KUKA KRL program: MyProgram_039().src

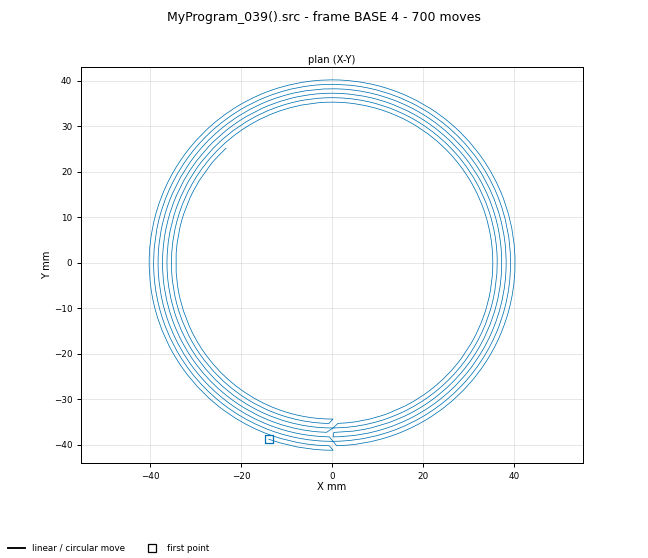
[picture p0: tool path of MyProgram_039().src in frame BASE 4, 700 of 700 moves have a stored position in this frame; points joined in program order, loops and branches not executed]
&ACCESS RVP
&REL 1
&PARAM TEMPLATE = C:\KRC\Roboter\Template\vorgabe
&PARAM EDITMASK = *
DEF MyProgram_039()
; ---- Setting reference (Base) ----
$BASE = BASE_DATA[4]

; --------------------------
; ---- Setting tool (TCP) ----
$TOOL = TOOL_DATA[3]
; --------------------------

$VEL.CP = VEL_APROX_PRINT
Startdeposition()
$VEL.CP = VEL_PRINT
LIN {X -13.9314,Y -38.786,Z 62,A -114.6314,B 24.865,C -2.6814,E1 24.9501,E2 -882.0703} C_DIS
LIN {X -11.5629,Y -39.5572,Z 62,A -111.3021,B 24.8654,C -2.6773,E1 24.959,E2 -885.3951} C_DIS
LIN {X -7.6518,Y -40.4959,Z 62,A -105.6604,B 24.8656,C -2.6755,E1 24.9744,E2 -891.0395} C_DIS
LIN {X -3.6812,Y -41.0476,Z 62,A -101.0464,B 24.867,C -2.6611,E1 24.9871,E2 -895.6225} C_DIS
LIN {X -1.5443,Y -41.1835,Z 62,A -97.4937,B 24.8662,C -2.6695,E1 24.9971,E2 -899.1962} C_DIS
LIN {X 0.2272,Y -41.2107,Z 62,A -96.0828,B 24.8676,C -2.6549,E1 25.0009,E2 -900.5723} C_DIS
Enddeposition()
LIN {X 0.2272,Y -41.2107,Z 62,A -96.0828,B 24.8676,C -2.6549,E1 25.0009,E2 -900.5723} C_DIS
Startdeposition()
$VEL.CP = VEL_PRINT
LIN {X -0.6478,Y -40.2271,Z 62,A -98.5489,B 24.8676,C -2.6549,E1 24.994,E2 -898.1063} C_DIS
LIN {X -3.2727,Y -40.0993,Z 62,A -101.3996,B 24.8664,C -2.6669,E1 24.9861,E2 -895.2829} C_DIS
LIN {X -5.4668,Y -39.8599,Z 62,A -105.2407,B 24.8673,C -2.6581,E1 24.9754,E2 -891.4182} C_DIS
LIN {X -7.661,Y -39.4965,Z 62,A -108.5221,B 24.8673,C -2.6577,E1 24.9664,E2 -888.1324} C_DIS
LIN {X -11.0904,Y -38.674,Z 62,A -112.7672,B 24.8661,C -2.6705,E1 24.955,E2 -883.9117} C_DIS
LIN {X -13.1876,Y -38.0098,Z 62,A -116.0642,B 24.8661,C -2.6708,E1 24.9462,E2 -880.6094} C_DIS
LIN {X -14.8236,Y -37.4023,Z 62,A -118.7522,B 24.8661,C -2.6705,E1 24.9392,E2 -877.915} C_DIS
LIN {X -16.9715,Y -36.4778,Z 62,A -122.3923,B 24.8661,C -2.6703,E1 24.9299,E2 -874.2655} C_DIS
LIN {X -19.0452,Y -35.4396,Z 62,A -125.8891,B 24.8659,C -2.6721,E1 24.9213,E2 -870.7634} C_DIS
LIN {X -21.3264,Y -34.1152,Z 62,A -129.5564,B 24.8653,C -2.6786,E1 24.9125,E2 -867.1001} C_DIS
LIN {X -23.9181,Y -32.3513,Z 62,A -133.265,B 24.8636,C -2.6947,E1 24.9041,E2 -863.4174} C_DIS
LIN {X -24.9832,Y -31.5356,Z 62,A -135.8558,B 24.8641,C -2.6902,E1 24.8984,E2 -860.8061} C_DIS
LIN {X -27.1159,Y -29.7221,Z 62,A -139.8787,B 24.8634,C -2.6974,E1 24.89,E2 -856.7844} C_DIS
LIN {X -29.6132,Y -27.2346,Z 62,A -145.2463,B 24.8627,C -2.7041,E1 24.8796,E2 -851.4096} C_DIS
LIN {X -31.9042,Y -24.511,Z 62,A -149.7729,B 24.8609,C -2.7217,E1 24.8717,E2 -846.904} C_DIS
LIN {X -33.4178,Y -22.404,Z 62,A -153.3459,B 24.8598,C -2.732,E1 24.866,E2 -843.3382} C_DIS
LIN {X -34.8539,Y -20.0965,Z 62,A -157.7346,B 24.8594,C -2.7364,E1 24.8596,E2 -838.9374} C_DIS
LIN {X -35.821,Y -18.3171,Z 62,A -160.6792,B 24.8586,C -2.7435,E1 24.8559,E2 -835.994} C_DIS
LIN {X -37.3884,Y -14.859,Z 62,A -165.4434,B 24.8564,C -2.7653,E1 24.8506,E2 -831.2557} C_DIS
LIN {X -38.3923,Y -12.0287,Z 62,A -169.7475,B 24.8551,C -2.7774,E1 24.8467,E2 -826.956} C_DIS
LIN {X -38.9921,Y -9.9139,Z 62,A -173.1815,B 24.8545,C -2.7835,E1 24.8442,E2 -823.5167} C_DIS
LIN {X -39.4343,Y -7.9754,Z 62,A -175.777,B 24.8533,C -2.7945,E1 24.8427,E2 -820.9322} C_DIS
LIN {X -39.7512,Y -6.2052,Z 62,A -178.4512,B 24.8526,C -2.8012,E1 24.8414,E2 -818.258} C_DIS
LIN {X -39.9928,Y -4.3853,Z 62,A 178.6144,B 24.8521,C -2.806,E1 24.8405,E2 -815.3176} C_DIS
LIN {X -40.2233,Y -0.8728,Z 62,A 173.9136,B 24.8501,C -2.8247,E1 24.8398,E2 -810.6334} C_DIS
LIN {X -40.2171,Y 1.1205,Z 62,A 170.9206,B 24.8493,C -2.8321,E1 24.8399,E2 -807.6399} C_DIS
LIN {X -40.0923,Y 3.3605,Z 62,A 167.875,B 24.8481,C -2.8436,E1 24.8405,E2 -804.6036} C_DIS
LIN {X -39.7922,Y 5.9355,Z 62,A 163.6374,B 24.8474,C -2.8496,E1 24.842,E2 -800.3551} C_DIS
LIN {X -39.2552,Y 8.8142,Z 62,A 159.4943,B 24.846,C -2.8629,E1 24.8444,E2 -796.2192} C_DIS
LIN {X -38.7278,Y 10.9006,Z 62,A 157.0034,B 24.8444,C -2.8781,E1 24.8461,E2 -793.7504} C_DIS
LIN {X -38.0306,Y 13.1284,Z 62,A 152.8289,B 24.8442,C -2.8795,E1 24.8498,E2 -789.5553} C_DIS
LIN {X -37.0608,Y 15.6577,Z 62,A 149.4783,B 24.8424,C -2.8962,E1 24.8533,E2 -786.226} C_DIS
LIN {X -36.1922,Y 17.5728,Z 62,A 146.5235,B 24.8414,C -2.9054,E1 24.8568,E2 -783.277} C_DIS
LIN {X -35.2767,Y 19.3455,Z 62,A 143.6101,B 24.8406,C -2.9127,E1 24.8606,E2 -780.3657} C_DIS
LIN {X -34.3469,Y 20.9512,Z 62,A 141.1264,B 24.8396,C -2.9218,E1 24.8641,E2 -777.8908} C_DIS
LIN {X -33.3523,Y 22.5009,Z 62,A 138.2963,B 24.839,C -2.9267,E1 24.8685,E2 -775.0583} C_DIS
LIN {X -32.3566,Y 23.9112,Z 62,A 136.0799,B 24.838,C -2.9358,E1 24.8721,E2 -772.8529} C_DIS
LIN {X -31.3616,Y 25.2019,Z 62,A 133.6236,B 24.8375,C -2.9403,E1 24.8763,E2 -770.3958} C_DIS
LIN {X -29.8637,Y 26.9597,Z 62,A 129.6067,B 24.8375,C -2.9407,E1 24.8838,E2 -766.3618} C_DIS
LIN {X -27.3552,Y 29.5017,Z 62,A 124.8309,B 24.8358,C -2.9559,E1 24.8933,E2 -761.6023} C_DIS
LIN {X -25.6158,Y 31.0243,Z 62,A 121.8887,B 24.8346,C -2.9669,E1 24.8995,E2 -758.6751} C_DIS
LIN {X -23.4742,Y 32.6748,Z 62,A 117.275,B 24.8346,C -2.9662,E1 24.9099,E2 -754.0432} C_DIS
LIN {X -21.3763,Y 34.084,Z 62,A 114.5678,B 24.8328,C -2.983,E1 24.9161,E2 -751.3674} C_DIS
LIN {X -19.8504,Y 34.9945,Z 62,A 111.4509,B 24.833,C -2.9806,E1 24.9237,E2 -748.2356} C_DIS
LIN {X -17.4004,Y 36.2751,Z 62,A 107.4729,B 24.8324,C -2.9864,E1 24.9336,E2 -744.2607} C_DIS
LIN {X -15.4532,Y 37.1467,Z 62,A 104.8887,B 24.8313,C -2.996,E1 24.9402,E2 -741.6935} C_DIS
LIN {X -14.0704,Y 37.6913,Z 62,A 102.6182,B 24.8312,C -2.9969,E1 24.9462,E2 -739.4204} C_DIS
LIN {X -11.8852,Y 38.437,Z 62,A 99.4969,B 24.8305,C -3.0027,E1 24.9544,E2 -736.3073} C_DIS
LIN {X -9.4063,Y 39.1174,Z 62,A 95.3264,B 24.8308,C -3.0001,E1 24.9657,E2 -732.1242} C_DIS
LIN {X -6.6101,Y 39.6859,Z 62,A 91.3009,B 24.8304,C -3.0036,E1 24.9768,E2 -728.1029} C_DIS
LIN {X -4.4808,Y 39.9828,Z 62,A 88.7069,B 24.8296,C -3.0113,E1 24.9839,E2 -725.5255} C_DIS
LIN {X -2.6075,Y 40.1481,Z 62,A 85.7171,B 24.8299,C -3.0085,E1 24.9922,E2 -722.5276} C_DIS
LIN {X -0.1087,Y 40.2327,Z 62,A 82.638,B 24.8291,C -3.0157,E1 25.0008,E2 -719.4655} C_DIS
LIN {X 1.836,Y 40.1908,Z 62,A 79.647,B 24.8294,C -3.013,E1 25.0092,E2 -716.4688} C_DIS
LIN {X 3.4769,Y 40.0827,Z 62,A 76.9649,B 24.8299,C -3.0084,E1 25.0166,E2 -713.7769} C_DIS
LIN {X 6.296,Y 39.7372,Z 62,A 72.7463,B 24.8303,C -3.0051,E1 25.0283,E2 -709.5541} C_DIS
LIN {X 8.6742,Y 39.2865,Z 62,A 69.7869,B 24.8297,C -3.0102,E1 25.0364,E2 -706.6107} C_DIS
LIN {X 10.2822,Y 38.8969,Z 62,A 67.448,B 24.8298,C -3.0091,E1 25.0427,E2 -704.2726} C_DIS
LIN {X 11.8652,Y 38.4432,Z 62,A 64.9198,B 24.8303,C -3.0049,E1 25.0495,E2 -701.7388} C_DIS
LIN {X 14.0198,Y 37.7116,Z 62,A 61.314,B 24.8312,C -2.9969,E1 25.059,E2 -698.1214} C_DIS
LIN {X 16.0999,Y 36.8708,Z 62,A 58.2555,B 24.8314,C -2.9955,E1 25.0668,E2 -695.0669} C_DIS
LIN {X 18.5215,Y 35.7165,Z 62,A 54.2669,B 24.8322,C -2.9883,E1 25.0768,E2 -691.0721} C_DIS
LIN {X 21.6163,Y 33.9325,Z 62,A 49.8972,B 24.8318,C -2.9916,E1 25.0872,E2 -686.7237} C_DIS
LIN {X 22.887,Y 33.0882,Z 62,A 47.2896,B 24.8329,C -2.9817,E1 25.0933,E2 -684.1013} C_DIS
LIN {X 24.9599,Y 31.5542,Z 62,A 43.6765,B 24.8335,C -2.9762,E1 25.1013,E2 -680.4883} C_DIS
LIN {X 27.0653,Y 29.7679,Z 62,A 39.822,B 24.8342,C -2.9698,E1 25.1094,E2 -676.634} C_DIS
LIN {X 28.2241,Y 28.6717,Z 62,A 37.3327,B 24.8351,C -2.9618,E1 25.1144,E2 -674.1361} C_DIS
LIN {X 30.1029,Y 26.6929,Z 62,A 33.4634,B 24.8361,C -2.9536,E1 25.1217,E2 -670.2645} C_DIS
LIN {X 32.3479,Y 23.9231,Z 62,A 29.2051,B 24.8359,C -2.9547,E1 25.129,E2 -666.0287} C_DIS
LIN {X 33.4895,Y 22.2968,Z 62,A 25.6289,B 24.838,C -2.9358,E1 25.1347,E2 -662.4254} C_DIS
LIN {X 34.8635,Y 20.0797,Z 62,A 22.1818,B 24.8386,C -2.9305,E1 25.1396,E2 -658.9834} C_DIS
LIN {X 36.1407,Y 17.6791,Z 62,A 18.8238,B 24.8389,C -2.9284,E1 25.1439,E2 -655.6382} C_DIS
LIN {X 37.0914,Y 15.585,Z 62,A 15.3545,B 24.8402,C -2.9162,E1 25.1479,E2 -652.1588} C_DIS
LIN {X 37.6444,Y 14.1974,Z 62,A 12.6022,B 24.842,C -2.8999,E1 25.1507,E2 -649.3834} C_DIS
LIN {X 38.7364,Y 10.8701,Z 62,A 8.1595,B 24.8426,C -2.8942,E1 25.1543,E2 -644.9523} C_DIS
LIN {X 39.4881,Y 7.6983,Z 62,A 2.9478,B 24.8451,C -2.8709,E1 25.1575,E2 -639.7158} C_DIS
LIN {X 40.0248,Y 4.0747,Z 62,A -2.6419,B 24.8475,C -2.8487,E1 25.1594,E2 -634.1066} C_DIS
LIN {X 40.2168,Y 1.1298,Z 62,A -6.2592,B 24.8479,C -2.8452,E1 25.1598,E2 -630.5024} C_DIS
LIN {X 40.1866,Y -1.9108,Z 62,A -10.1736,B 24.8486,C -2.8385,E1 25.1595,E2 -626.5955} C_DIS
LIN {X 39.973,Y -4.5641,Z 62,A -14.341,B 24.8506,C -2.8204,E1 25.1584,E2 -622.4098} C_DIS
LIN {X 39.5912,Y -7.1552,Z 62,A -17.6584,B 24.8511,C -2.8155,E1 25.1569,E2 -619.1005} C_DIS
LIN {X 39.1774,Y -9.1541,Z 62,A -20.3468,B 24.8517,C -2.8101,E1 25.1553,E2 -616.415} C_DIS
LIN {X 38.7929,Y -10.6678,Z 62,A -22.4858,B 24.8522,C -2.8047,E1 25.1538,E2 -614.2753} C_DIS
LIN {X 38.435,Y -11.8916,Z 62,A -24.5159,B 24.8532,C -2.7956,E1 25.1521,E2 -612.2352} C_DIS
LIN {X 37.8279,Y -13.7011,Z 62,A -27.1869,B 24.854,C -2.7881,E1 25.1496,E2 -609.5616} C_DIS
LIN {X 37.1317,Y -15.4894,Z 62,A -29.7821,B 24.8546,C -2.7822,E1 25.1469,E2 -606.9669} C_DIS
LIN {X 36.5158,Y -16.8898,Z 62,A -31.9189,B 24.8552,C -2.7765,E1 25.1445,E2 -604.828} C_DIS
LIN {X 35.8809,Y -18.1999,Z 62,A -34.1771,B 24.8562,C -2.7674,E1 25.1417,E2 -602.5605} C_DIS
LIN {X 34.932,Y -19.9598,Z 62,A -36.8662,B 24.8567,C -2.7619,E1 25.138,E2 -599.8724} C_DIS
LIN {X 34.0278,Y -21.4662,Z 62,A -39.4907,B 24.8577,C -2.7529,E1 25.1342,E2 -597.2399} C_DIS
LIN {X 32.8611,Y -23.213,Z 62,A -42.6003,B 24.8587,C -2.7429,E1 25.1293,E2 -594.1218} C_DIS
LIN {X 31.0693,Y -25.5616,Z 62,A -46.6066,B 24.8595,C -2.7351,E1 25.1224,E2 -590.1162} C_DIS
LIN {X 28.8552,Y -28.0355,Z 62,A -51.8146,B 24.8615,C -2.7159,E1 25.1124,E2 -584.8854} C_DIS
LIN {X 26.4064,Y -30.354,Z 62,A -56.7712,B 24.8628,C -2.7026,E1 25.1022,E2 -579.9173} C_DIS
LIN {X 24.1954,Y -32.1442,Z 62,A -59.8338,B 24.8621,C -2.7095,E1 25.0955,E2 -576.8823} C_DIS
LIN {X 21.917,Y -33.7395,Z 62,A -63.7114,B 24.8628,C -2.703,E1 25.0866,E2 -573.0025} C_DIS
LIN {X 20.486,Y -34.6263,Z 62,A -66.5733,B 24.864,C -2.6915,E1 25.0797,E2 -570.1223} C_DIS
LIN {X 18.9049,Y -35.5148,Z 62,A -68.867,B 24.864,C -2.6915,E1 25.0741,E2 -567.8352} C_DIS
LIN {X 17.2843,Y -36.3309,Z 62,A -71.6851,B 24.8647,C -2.6838,E1 25.067,E2 -565.0066} C_DIS
LIN {X 15.5388,Y -37.1109,Z 62,A -74.2668,B 24.8649,C -2.682,E1 25.0604,E2 -562.4266} C_DIS
LIN {X 14.1244,Y -37.672,Z 62,A -76.2369,B 24.8649,C -2.682,E1 25.0553,E2 -560.4609} C_DIS
LIN {X 12.7445,Y -38.1608,Z 62,A -78.418,B 24.8653,C -2.678,E1 25.0495,E2 -558.2746} C_DIS
LIN {X 10.8494,Y -38.7423,Z 62,A -81.6556,B 24.8662,C -2.6688,E1 25.0408,E2 -555.0209} C_DIS
LIN {X 8.35,Y -39.3566,Z 62,A -85.5356,B 24.8669,C -2.6624,E1 25.0302,E2 -551.1308} C_DIS
LIN {X 5.1609,Y -39.9002,Z 62,A -89.5422,B 24.8664,C -2.6677,E1 25.0192,E2 -547.1406} C_DIS
LIN {X 3.4473,Y -40.0848,Z 62,A -92.3148,B 24.8669,C -2.6619,E1 25.0115,E2 -544.356} C_DIS
LIN {X 0.9853,Y -40.2212,Z 62,A -96.0879,B 24.8674,C -2.6571,E1 25.0009,E2 -540.5724} C_DIS
LIN {X 0.9853,Y -40.2212,Z 62,A -96.0879,B 24.8674,C -2.6571,E1 25.0009,E2 -540.5724} C_DIS
Enddeposition()
LIN {X 0.2181,Y -39.2481,Z 62,A -96.0532,B 24.8642,C -2.6894,E1 25.0012,E2 -540.6839} C_DIS
Startdeposition()
$VEL.CP = VEL_PRINT
LIN {X 1.643,Y -39.2185,Z 62,A -93.4048,B 24.8633,C -2.6978,E1 25.0087,E2 -543.3516} C_DIS
LIN {X 3.7925,Y -39.0693,Z 62,A -89.9922,B 24.8628,C -2.703,E1 25.0182,E2 -546.775} C_DIS
LIN {X 6.7082,Y -38.675,Z 62,A -85.0967,B 24.8616,C -2.7147,E1 25.0317,E2 -551.6934} C_DIS
LIN {X 9.6984,Y -38.0355,Z 62,A -81.1674,B 24.862,C -2.7111,E1 25.0424,E2 -555.6087} C_DIS
LIN {X 12.2339,Y -37.2976,Z 62,A -77.5539,B 24.8619,C -2.712,E1 25.052,E2 -559.2177} C_DIS
LIN {X 14.021,Y -36.6636,Z 62,A -74.6805,B 24.8613,C -2.7171,E1 25.0596,E2 -562.0973} C_DIS
LIN {X 15.991,Y -35.8483,Z 62,A -71.4397,B 24.8607,C -2.7236,E1 25.0679,E2 -565.3456} C_DIS
LIN {X 18.5513,Y -34.593,Z 62,A -67.5163,B 24.8604,C -2.7267,E1 25.0776,E2 -569.2657} C_DIS
LIN {X 20.4377,Y -33.5126,Z 62,A -64.3458,B 24.8598,C -2.7324,E1 25.0853,E2 -572.4399} C_DIS
LIN {X 22.1696,Y -32.3934,Z 62,A -61.2775,B 24.8591,C -2.7391,E1 25.0924,E2 -575.5138} C_DIS
LIN {X 23.8623,Y -31.1672,Z 62,A -58.4305,B 24.8588,C -2.7421,E1 25.0988,E2 -578.3579} C_DIS
LIN {X 25.1855,Y -30.1071,Z 62,A -55.7668,B 24.8579,C -2.7505,E1 25.1045,E2 -581.0312} C_DIS
LIN {X 26.9367,Y -28.5519,Z 62,A -52.347,B 24.8571,C -2.7583,E1 25.1116,E2 -584.4557} C_DIS
LIN {X 28.6666,Y -26.8146,Z 62,A -49.0657,B 24.8567,C -2.7622,E1 25.118,E2 -587.732} C_DIS
LIN {X 29.783,Y -25.5692,Z 62,A -46.5538,B 24.8559,C -2.7694,E1 25.1226,E2 -590.2498} C_DIS
LIN {X 31.0822,Y -23.9727,Z 62,A -43.4403,B 24.8549,C -2.779,E1 25.128,E2 -593.3714} C_DIS
LIN {X 32.1373,Y -22.5392,Z 62,A -41.0856,B 24.8546,C -2.782,E1 25.1318,E2 -595.7218} C_DIS
LIN {X 33.3027,Y -20.778,Z 62,A -38.0289,B 24.8538,C -2.79,E1 25.1365,E2 -598.7823} C_DIS
LIN {X 34.3602,Y -18.9783,Z 62,A -34.6531,B 24.8523,C -2.804,E1 25.1412,E2 -602.1737} C_DIS
LIN {X 35.3413,Y -17.0819,Z 62,A -31.7247,B 24.8517,C -2.81,E1 25.1448,E2 -605.1006} C_DIS
LIN {X 36.2028,Y -15.1708,Z 62,A -28.8924,B 24.8511,C -2.8153,E1 25.148,E2 -607.93} C_DIS
LIN {X 36.7141,Y -13.8877,Z 62,A -26.4345,B 24.8497,C -2.8287,E1 25.1505,E2 -610.4059} C_DIS
LIN {X 37.6399,Y -11.1369,Z 62,A -22.7022,B 24.8492,C -2.8332,E1 25.1536,E2 -614.1278} C_DIS
LIN {X 38.2954,Y -8.6166,Z 62,A -18.2157,B 24.8467,C -2.8564,E1 25.1566,E2 -618.6432} C_DIS
LIN {X 38.7766,Y -6.0971,Z 62,A -15.0431,B 24.8465,C -2.8586,E1 25.1581,E2 -621.8023} C_DIS
LIN {X 39.0542,Y -3.9454,Z 62,A -11.7449,B 24.8452,C -2.8707,E1 25.1592,E2 -625.1097} C_DIS
LIN {X 39.2374,Y -1.1094,Z 62,A -7.052,B 24.8428,C -2.8928,E1 25.1598,E2 -629.827} C_DIS
LIN {X 39.2044,Y 1.954,Z 62,A -2.7533,B 24.8416,C -2.9039,E1 25.1594,E2 -634.1263} C_DIS
LIN {X 38.8443,Y 5.6508,Z 62,A 2.8909,B 24.8393,C -2.9243,E1 25.1574,E2 -639.7855} C_DIS
LIN {X 38.0551,Y 9.6239,Z 62,A 7.4821,B 24.8397,C -2.9203,E1 25.1548,E2 -644.3406} C_DIS
LIN {X 37.2758,Y 12.3016,Z 62,A 12.1812,B 24.8373,C -2.9425,E1 25.1509,E2 -649.0654} C_DIS
LIN {X 36.5171,Y 14.3977,Z 62,A 15.3004,B 24.8365,C -2.9496,E1 25.1479,E2 -652.1841} C_DIS
LIN {X 35.8241,Y 16.0446,Z 62,A 17.8534,B 24.8358,C -2.956,E1 25.145,E2 -654.7383} C_DIS
LIN {X 34.6303,Y 18.4816,Z 62,A 22.0919,B 24.8341,C -2.9711,E1 25.1396,E2 -658.9902} C_DIS
LIN {X 33.7687,Y 20.0117,Z 62,A 24.6893,B 24.8333,C -2.9783,E1 25.1359,E2 -661.5913} C_DIS
LIN {X 32.3499,Y 22.2315,Z 62,A 28.2911,B 24.8326,C -2.9841,E1 25.1304,E2 -665.1887} C_DIS
LIN {X 31.3754,Y 23.5876,Z 62,A 31.02,B 24.8315,C -2.9945,E1 25.1258,E2 -667.9293} C_DIS
LIN {X 29.4047,Y 26.0041,Z 62,A 35.0326,B 24.8313,C -2.9963,E1 25.1186,E2 -671.9279} C_DIS
LIN {X 27.9864,Y 27.5239,Z 62,A 38.3392,B 24.8301,C -3.007,E1 25.1122,E2 -675.2455} C_DIS
LIN {X 25.8182,Y 29.567,Z 62,A 42.4929,B 24.8294,C -3.0125,E1 25.1036,E2 -679.3955} C_DIS
LIN {X 24.2569,Y 30.861,Z 62,A 45.6484,B 24.8285,C -3.0208,E1 25.0967,E2 -682.5589} C_DIS
LIN {X 21.9802,Y 32.5217,Z 62,A 49.3111,B 24.8285,C -3.0208,E1 25.0884,E2 -686.2088} C_DIS
LIN {X 20.7805,Y 33.3011,Z 62,A 51.585,B 24.8278,C -3.0268,E1 25.0831,E2 -688.4895} C_DIS
LIN {X 19.1084,Y 34.2876,Z 62,A 54.4953,B 24.8272,C -3.0318,E1 25.076,E2 -691.403} C_DIS
LIN {X 17.737,Y 35.0173,Z 62,A 56.9423,B 24.8266,C -3.0372,E1 25.0699,E2 -693.8563} C_DIS
LIN {X 15.0204,Y 36.2662,Z 62,A 61.2608,B 24.8261,C -3.0413,E1 25.0588,E2 -698.1738} C_DIS
LIN {X 12.6571,Y 37.1565,Z 62,A 65.1095,B 24.8255,C -3.0468,E1 25.0487,E2 -702.0277} C_DIS
LIN {X 9.6817,Y 38.0403,Z 62,A 69.4045,B 24.8255,C -3.0464,E1 25.0372,E2 -706.3149} C_DIS
LIN {X 7.7562,Y 38.4793,Z 62,A 71.9499,B 24.8259,C -3.0431,E1 25.0303,E2 -708.8491} C_DIS
LIN {X 5.9682,Y 38.7966,Z 62,A 74.7741,B 24.8256,C -3.0463,E1 25.0225,E2 -711.6781} C_DIS
LIN {X 4.0502,Y 39.0434,Z 62,A 77.8312,B 24.8251,C -3.0499,E1 25.014,E2 -714.7416} C_DIS
LIN {X 0.6187,Y 39.2482,Z 62,A 82.5353,B 24.8257,C -3.0455,E1 25.0009,E2 -719.4336} C_DIS
LIN {X -1.391,Y 39.2287,Z 62,A 85.6323,B 24.8255,C -3.0468,E1 24.9922,E2 -722.5342} C_DIS
LIN {X -3.5836,Y 39.089,Z 62,A 88.5093,B 24.8261,C -3.0412,E1 24.9842,E2 -725.3991} C_DIS
LIN {X -6.1003,Y 38.7758,Z 62,A 92.8808,B 24.8254,C -3.0474,E1 24.9721,E2 -729.7888} C_DIS
LIN {X -8.9337,Y 38.2229,Z 62,A 96.9696,B 24.826,C -3.0423,E1 24.961,E2 -733.8703} C_DIS
LIN {X -11.0142,Y 37.6763,Z 62,A 99.6454,B 24.827,C -3.0334,E1 24.9538,E2 -736.529} C_DIS
LIN {X -13.4567,Y 36.8742,Z 62,A 104.3487,B 24.8262,C -3.0403,E1 24.9413,E2 -741.2581} C_DIS
LIN {X -15.918,Y 35.8812,Z 62,A 108.0064,B 24.8272,C -3.0322,E1 24.932,E2 -744.905} C_DIS
LIN {X -18.8632,Y 34.4236,Z 62,A 112.1034,B 24.829,C -3.0163,E1 24.9219,E2 -748.9753} C_DIS
LIN {X -20.1405,Y 33.6926,Z 62,A 114.631,B 24.829,C -3.0169,E1 24.9158,E2 -751.5119} C_DIS
LIN {X -22.1342,Y 32.417,Z 62,A 118.1436,B 24.8296,C -3.0111,E1 24.9076,E2 -755.022} C_DIS
LIN {X -24.2708,Y 30.8501,Z 62,A 121.8413,B 24.8307,C -3.0012,E1 24.8994,E2 -758.7096} C_DIS
LIN {X -25.9398,Y 29.4609,Z 62,A 124.7274,B 24.8318,C -2.9912,E1 24.8933,E2 -761.583} C_DIS
LIN {X -26.9008,Y 28.5856,Z 62,A 126.6875,B 24.8322,C -2.9876,E1 24.8893,E2 -763.5423} C_DIS
LIN {X -27.9619,Y 27.5486,Z 62,A 128.9001,B 24.8328,C -2.983,E1 24.8849,E2 -765.7533} C_DIS
LIN {X -29.0381,Y 26.4117,Z 62,A 131.5109,B 24.833,C -2.981,E1 24.88,E2 -768.3707} C_DIS
LIN {X -30.5442,Y 24.6546,Z 62,A 134.8511,B 24.834,C -2.972,E1 24.874,E2 -771.7049} C_DIS
LIN {X -31.5157,Y 23.4008,Z 62,A 137.298,B 24.8345,C -2.9674,E1 24.8699,E2 -774.1524} C_DIS
LIN {X -32.6143,Y 21.8421,Z 62,A 140.126,B 24.8353,C -2.9604,E1 24.8655,E2 -776.9777} C_DIS
LIN {X -34.0401,Y 19.5464,Z 62,A 143.9029,B 24.8367,C -2.9476,E1 24.8601,E2 -780.7435} C_DIS
LIN {X -35.0735,Y 17.6264,Z 62,A 147.1653,B 24.8376,C -2.9393,E1 24.8559,E2 -784.0035} C_DIS
LIN {X -35.8401,Y 16.0092,Z 62,A 149.6138,B 24.8387,C -2.93,E1 24.853,E2 -786.443} C_DIS
LIN {X -36.6628,Y 14.023,Z 62,A 153.2305,B 24.8392,C -2.9255,E1 24.8493,E2 -790.0694} C_DIS
LIN {X -37.589,Y 11.3086,Z 62,A 157.0632,B 24.841,C -2.9092,E1 24.846,E2 -793.8849} C_DIS
LIN {X -38.108,Y 9.4101,Z 62,A 160.0554,B 24.8418,C -2.9016,E1 24.8439,E2 -796.8763} C_DIS
LIN {X -38.5678,Y 7.3029,Z 62,A 163.8033,B 24.8422,C -2.8979,E1 24.8419,E2 -800.6376} C_DIS
LIN {X -39.1208,Y 3.2194,Z 62,A 169.7039,B 24.8444,C -2.8779,E1 24.8401,E2 -806.5255} C_DIS
LIN {X -39.2526,Y 0.1735,Z 62,A 173.3655,B 24.8468,C -2.8559,E1 24.8398,E2 -810.1567} C_DIS
LIN {X -39.2383,Y -1.0798,Z 62,A 175.4373,B 24.8471,C -2.8527,E1 24.8398,E2 -812.2331} C_DIS
LIN {X -39.1527,Y -2.8074,Z 62,A 177.9946,B 24.8479,C -2.8451,E1 24.8403,E2 -814.7878} C_DIS
LIN {X -38.9868,Y -4.5629,Z 62,A -179.3903,B 24.8487,C -2.8376,E1 24.8411,E2 -817.4006} C_DIS
LIN {X -38.7368,Y -6.3455,Z 62,A -176.5464,B 24.8493,C -2.8318,E1 24.8423,E2 -820.2475} C_DIS
LIN {X -38.3097,Y -8.5554,Z 62,A -173.4141,B 24.8506,C -2.8203,E1 24.8441,E2 -823.3707} C_DIS
LIN {X -37.8399,Y -10.4391,Z 62,A -170.5824,B 24.8515,C -2.8119,E1 24.8461,E2 -826.1987} C_DIS
LIN {X -37.282,Y -12.2837,Z 62,A -167.5843,B 24.8521,C -2.8056,E1 24.8486,E2 -829.199} C_DIS
LIN {X -36.6851,Y -13.9644,Z 62,A -164.5988,B 24.8525,C -2.8022,E1 24.8516,E2 -832.1932} C_DIS
LIN {X -35.6074,Y -16.52,Z 62,A -160.6536,B 24.8538,C -2.7899,E1 24.856,E2 -836.1306} C_DIS
LIN {X -34.0847,Y -19.4688,Z 62,A -155.6676,B 24.855,C -2.7785,E1 24.8627,E2 -841.1159} C_DIS
LIN {X -33.0991,Y -21.101,Z 62,A -153.0725,B 24.8559,C -2.7694,E1 24.8665,E2 -843.7025} C_DIS
LIN {X -31.7594,Y -23.0685,Z 62,A -149.8699,B 24.8571,C -2.758,E1 24.8716,E2 -846.8934} C_DIS
LIN {X -30.427,Y -24.7992,Z 62,A -146.3384,B 24.8575,C -2.7544,E1 24.8778,E2 -850.433} C_DIS
LIN {X -28.9153,Y -26.5461,Z 62,A -143.2985,B 24.8586,C -2.7433,E1 24.8834,E2 -853.4599} C_DIS
LIN {X -27.3276,Y -28.1782,Z 62,A -139.7112,B 24.859,C -2.7395,E1 24.8905,E2 -857.0532} C_DIS
LIN {X -25.6321,Y -29.729,Z 62,A -136.3978,B 24.8598,C -2.7326,E1 24.8974,E2 -860.3633} C_DIS
LIN {X -24.249,Y -30.8673,Z 62,A -134.1053,B 24.8606,C -2.7242,E1 24.9024,E2 -862.6444} C_DIS
LIN {X -22.8087,Y -31.9461,Z 62,A -131.1987,B 24.8607,C -2.7231,E1 24.909,E2 -865.5585} C_DIS
LIN {X -20.9161,Y -33.2164,Z 62,A -128.1769,B 24.8616,C -2.7144,E1 24.916,E2 -868.5694} C_DIS
LIN {X -19.2206,Y -34.2253,Z 62,A -124.6587,B 24.8612,C -2.7181,E1 24.9246,E2 -872.107} C_DIS
LIN {X -16.7678,Y -35.492,Z 62,A -120.8058,B 24.862,C -2.7112,E1 24.9342,E2 -875.9535} C_DIS
LIN {X -14.4586,Y -36.4932,Z 62,A -117.8418,B 24.8632,C -2.6987,E1 24.9417,E2 -878.8945} C_DIS
LIN {X -12.6931,Y -37.1442,Z 62,A -114.3739,B 24.8625,C -2.7054,E1 24.9509,E2 -882.3853} C_DIS
LIN {X -10.9024,Y -37.7091,Z 62,A -112.007,B 24.8632,C -2.6988,E1 24.9572,E2 -884.7404} C_DIS
LIN {X -9.0524,Y -38.1955,Z 62,A -108.8167,B 24.8628,C -2.7024,E1 24.9659,E2 -887.9438} C_DIS
LIN {X -7.0512,Y -38.6146,Z 62,A -106.0922,B 24.8633,C -2.6979,E1 24.9733,E2 -890.6606} C_DIS
LIN {X -5.132,Y -38.9161,Z 62,A -102.701,B 24.8626,C -2.7047,E1 24.9828,E2 -894.0707} C_DIS
LIN {X -2.8769,Y -39.148,Z 62,A -100.0324,B 24.8635,C -2.6959,E1 24.9901,E2 -896.7197} C_DIS
LIN {X -1.5857,Y -39.2207,Z 62,A -97.848,B 24.8631,C -2.7001,E1 24.9963,E2 -898.9146} C_DIS
LIN {X 0.2181,Y -39.2481,Z 62,A -96.053,B 24.8642,C -2.6893,E1 25.0012,E2 -900.6839} C_DIS
Enddeposition()
LIN {X 0.2181,Y -39.2481,Z 62,A -96.053,B 24.8642,C -2.6893,E1 25.0012,E2 -900.6839} C_DIS
Startdeposition()
$VEL.CP = VEL_PRINT
LIN {X -0.6151,Y -38.2682,Z 62,A -98.0809,B 24.8635,C -2.6957,E1 24.9956,E2 -898.6711} C_DIS
LIN {X -2.7121,Y -38.1773,Z 62,A -101.1684,B 24.8635,C -2.6962,E1 24.987,E2 -895.584} C_DIS
LIN {X -4.6452,Y -37.9908,Z 62,A -104.1189,B 24.8635,C -2.696,E1 24.9788,E2 -892.6312} C_DIS
LIN {X -6.4062,Y -37.7335,Z 62,A -106.6893,B 24.8633,C -2.6979,E1 24.9717,E2 -890.063} C_DIS
LIN {X -8.0495,Y -37.4174,Z 62,A -109.0793,B 24.8631,C -2.7003,E1 24.9652,E2 -887.676} C_DIS
LIN {X -9.4713,Y -37.0829,Z 62,A -111.4567,B 24.8631,C -2.6991,E1 24.9587,E2 -885.2924} C_DIS
LIN {X -11.3054,Y -36.5654,Z 62,A -114.324,B 24.8631,C -2.7009,E1 24.951,E2 -882.4245} C_DIS
LIN {X -13.2882,Y -35.8925,Z 62,A -117.2698,B 24.8625,C -2.7057,E1 24.9433,E2 -879.4845} C_DIS
LIN {X -14.91,Y -35.2496,Z 62,A -120.1156,B 24.8625,C -2.7055,E1 24.9359,E2 -876.6318} C_DIS
LIN {X -16.9314,Y -34.3246,Z 62,A -123.3874,B 24.8621,C -2.7099,E1 24.9277,E2 -873.3623} C_DIS
LIN {X -18.9249,Y -33.2674,Z 62,A -127.0108,B 24.8619,C -2.7116,E1 24.9188,E2 -869.7324} C_DIS
LIN {X -20.5483,Y -32.2895,Z 62,A -129.462,B 24.861,C -2.7201,E1 24.913,E2 -867.2937} C_DIS
LIN {X -21.6871,Y -31.5365,Z 62,A -131.6238,B 24.8609,C -2.7219,E1 24.908,E2 -865.1292} C_DIS
LIN {X -22.9868,Y -30.6015,Z 62,A -134.1052,B 24.8605,C -2.725,E1 24.9024,E2 -862.6464} C_DIS
LIN {X -24.5266,Y -29.3819,Z 62,A -136.923,B 24.8599,C -2.7317,E1 24.8963,E2 -859.8338} C_DIS
LIN {X -25.7185,Y -28.3451,Z 62,A -139.4163,B 24.8595,C -2.7348,E1 24.8911,E2 -857.3381} C_DIS
LIN {X -27.0972,Y -27.029,Z 62,A -142.1373,B 24.8588,C -2.742,E1 24.8857,E2 -854.623} C_DIS
LIN {X -28.2175,Y -25.8576,Z 62,A -144.6538,B 24.8584,C -2.7462,E1 24.8809,E2 -852.1056} C_DIS
LIN {X -29.3495,Y -24.5649,Z 62,A -147.2405,B 24.8578,C -2.7518,E1 24.8762,E2 -849.5204} C_DIS
LIN {X -30.4976,Y -23.125,Z 62,A -149.91,B 24.857,C -2.7591,E1 24.8716,E2 -846.8558} C_DIS
LIN {X -31.3176,Y -22.0015,Z 62,A -152.4735,B 24.857,C -2.7592,E1 24.8674,E2 -844.28} C_DIS
LIN {X -32.5375,Y -20.1538,Z 62,A -155.8455,B 24.8562,C -2.767,E1 24.8624,E2 -840.9096} C_DIS
LIN {X -33.9355,Y -17.6989,Z 62,A -159.7086,B 24.8546,C -2.7819,E1 24.8572,E2 -837.0615} C_DIS
LIN {X -34.9905,Y -15.5097,Z 62,A -163.9265,B 24.8542,C -2.7861,E1 24.8522,E2 -832.8308} C_DIS
LIN {X -35.8349,Y -13.443,Z 62,A -166.6638,B 24.8526,C -2.8015,E1 24.8495,E2 -830.115} C_DIS
LIN {X -36.3843,Y -11.8757,Z 62,A -169.1656,B 24.8518,C -2.8086,E1 24.8472,E2 -827.6159} C_DIS
LIN {X -36.8372,Y -10.3858,Z 62,A -171.4867,B 24.8511,C -2.8155,E1 24.8454,E2 -825.2979} C_DIS
LIN {X -37.2026,Y -8.99,Z 62,A -173.535,B 24.8503,C -2.823,E1 24.844,E2 -823.2557} C_DIS
LIN {X -37.588,Y -7.2101,Z 62,A -177.0262,B 24.8502,C -2.8239,E1 24.8421,E2 -819.746} C_DIS
LIN {X -38.07,Y -3.9396,Z 62,A 178.215,B 24.8484,C -2.841,E1 24.8404,E2 -814.9996} C_DIS
LIN {X -38.2213,Y -1.998,Z 62,A 175.6928,B 24.847,C -2.8538,E1 24.8399,E2 -812.4928} C_DIS
LIN {X -38.271,Y -0.4703,Z 62,A 173.3075,B 24.8463,C -2.86,E1 24.8398,E2 -810.108} C_DIS
LIN {X -38.2552,Y 1.1774,Z 62,A 170.7443,B 24.8456,C -2.8668,E1 24.8399,E2 -807.5457} C_DIS
LIN {X -38.1593,Y 2.9528,Z 62,A 168.215,B 24.8445,C -2.8764,E1 24.8404,E2 -805.0241} C_DIS
LIN {X -38.0327,Y 4.2871,Z 62,A 165.6747,B 24.8445,C -2.8776,E1 24.8411,E2 -802.4715} C_DIS
LIN {X -37.6092,Y 7.0999,Z 62,A 161.8935,B 24.8425,C -2.8954,E1 24.8429,E2 -798.7105} C_DIS
LIN {X -37.3085,Y 8.538,Z 62,A 159.297,B 24.8421,C -2.8985,E1 24.8444,E2 -796.106} C_DIS
LIN {X -36.6275,Y 11.1049,Z 62,A 155.5219,B 24.8406,C -2.9125,E1 24.8473,E2 -792.3427} C_DIS
LIN {X -35.996,Y 13.0055,Z 62,A 152.3846,B 24.8398,C -2.9203,E1 24.8501,E2 -789.2061} C_DIS
LIN {X -35.1968,Y 15.0355,Z 62,A 148.4472,B 24.8394,C -2.9235,E1 24.8544,E2 -785.2547} C_DIS
LIN {X -33.3206,Y 18.8314,Z 62,A 142.1058,B 24.8374,C -2.9417,E1 24.8626,E2 -778.9229} C_DIS
LIN {X -31.2784,Y 22.0558,Z 62,A 136.8927,B 24.8351,C -2.9621,E1 24.8706,E2 -773.7326} C_DIS
LIN {X -29.9487,Y 23.8314,Z 62,A 133.7584,B 24.8339,C -2.9726,E1 24.8759,E2 -770.6085} C_DIS
LIN {X -28.6344,Y 25.3958,Z 62,A 130.5849,B 24.8332,C -2.9791,E1 24.8817,E2 -767.436} C_DIS
LIN {X -27.2845,Y 26.8403,Z 62,A 127.6471,B 24.8324,C -2.9864,E1 24.8874,E2 -764.503} C_DIS
LIN {X -25.7927,Y 28.2769,Z 62,A 124.6219,B 24.8315,C -2.9942,E1 24.8935,E2 -761.4842} C_DIS
LIN {X -24.3513,Y 29.5276,Z 62,A 121.6784,B 24.8309,C -2.9995,E1 24.8998,E2 -758.5419} C_DIS
LIN {X -22.9732,Y 30.6117,Z 62,A 119.2445,B 24.8301,C -3.007,E1 24.9052,E2 -756.1169} C_DIS
LIN {X -21.009,Y 31.9917,Z 62,A 114.667,B 24.8305,C -3.0034,E1 24.9158,E2 -751.5156} C_DIS
LIN {X -18.1462,Y 33.6982,Z 62,A 110.0561,B 24.829,C -3.016,E1 24.927,E2 -746.9214} C_DIS
LIN {X -15.4426,Y 35.02,Z 62,A 106.053,B 24.8276,C -3.0283,E1 24.937,E2 -742.9376} C_DIS
LIN {X -14.1087,Y 35.5781,Z 62,A 103.9466,B 24.8272,C -3.0319,E1 24.9424,E2 -740.8351} C_DIS
LIN {X -12.4947,Y 36.1767,Z 62,A 101.1046,B 24.8272,C -3.0321,E1 24.9499,E2 -737.9878} C_DIS
LIN {X -10.5006,Y 36.8047,Z 62,A 97.9021,B 24.8269,C -3.0347,E1 24.9585,E2 -734.786} C_DIS
LIN {X -8.4564,Y 37.3275,Z 62,A 94.8606,B 24.8264,C -3.039,E1 24.9667,E2 -731.7506} C_DIS
LIN {X -5.7067,Y 37.8453,Z 62,A 89.6608,B 24.8274,C -3.03,E1 24.9811,E2 -726.5245} C_DIS
LIN {X -1.8109,Y 38.2308,Z 62,A 84.484,B 24.8262,C -3.0407,E1 24.9955,E2 -721.3712} C_DIS
LIN {X 0.8024,Y 38.265,Z 62,A 80.9102,B 24.8256,C -3.0457,E1 25.0054,E2 -717.8093} C_DIS
LIN {X 2.5355,Y 38.1892,Z 62,A 78.4216,B 24.8255,C -3.0471,E1 25.0123,E2 -715.3251} C_DIS
LIN {X 4.1446,Y 38.0481,Z 62,A 75.8556,B 24.8257,C -3.045,E1 25.0195,E2 -712.7555} C_DIS
LIN {X 6.1579,Y 37.7748,Z 62,A 72.6801,B 24.826,C -3.0424,E1 25.0283,E2 -709.5769} C_DIS
LIN {X 8.2637,Y 37.3707,Z 62,A 69.597,B 24.826,C -3.0427,E1 25.0367,E2 -706.4981} C_DIS
LIN {X 10.2661,Y 36.8708,Z 62,A 66.6798,B 24.826,C -3.0431,E1 25.0445,E2 -703.5865} C_DIS
LIN {X 12.5898,Y 36.1434,Z 62,A 62.7728,B 24.8267,C -3.0367,E1 25.0549,E2 -699.6717} C_DIS
LIN {X 14.1675,Y 35.5551,Z 62,A 60.214,B 24.827,C -3.0338,E1 25.0616,E2 -697.1116} C_DIS
LIN {X 16.1269,Y 34.7097,Z 62,A 57.4057,B 24.8268,C -3.0356,E1 25.0687,E2 -694.3146} C_DIS
LIN {X 17.4587,Y 34.0594,Z 62,A 55.2337,B 24.827,C -3.0335,E1 25.0742,E2 -692.1435} C_DIS
LIN {X 18.8343,Y 33.3188,Z 62,A 52.6443,B 24.8278,C -3.0269,E1 25.0805,E2 -689.5458} C_DIS
LIN {X 20.1104,Y 32.5646,Z 62,A 50.6212,B 24.8278,C -3.0264,E1 25.0853,E2 -687.5279} C_DIS
LIN {X 21.2211,Y 31.8518,Z 62,A 48.6371,B 24.8282,C -3.0233,E1 25.09,E2 -685.5429} C_DIS
LIN {X 22.7101,Y 30.8074,Z 62,A 45.6886,B 24.8291,C -3.0155,E1 25.0967,E2 -682.5863} C_DIS
LIN {X 24.623,Y 29.3011,Z 62,A 41.6667,B 24.8305,C -3.0034,E1 25.1054,E2 -678.551} C_DIS
LIN {X 26.6432,Y 27.4771,Z 62,A 37.5774,B 24.8314,C -2.9951,E1 25.1137,E2 -674.4586} C_DIS
LIN {X 28.7056,Y 25.3153,Z 62,A 33.4386,B 24.8319,C -2.9903,E1 25.1216,E2 -670.3267} C_DIS
LIN {X 30.3009,Y 23.3816,Z 62,A 29.7942,B 24.8327,C -2.9833,E1 25.1279,E2 -666.6827} C_DIS
LIN {X 31.8183,Y 21.2717,Z 62,A 25.5603,B 24.8344,C -2.9685,E1 25.1347,E2 -662.4346} C_DIS
LIN {X 32.9891,Y 19.4053,Z 62,A 22.1302,B 24.8356,C -2.958,E1 25.1396,E2 -658.9971} C_DIS
LIN {X 34.661,Y 16.2317,Z 62,A 17.264,B 24.8363,C -2.9512,E1 25.1457,E2 -654.1408} C_DIS
LIN {X 35.6192,Y 14.0041,Z 62,A 13.3072,B 24.838,C -2.9359,E1 25.1499,E2 -650.1695} C_DIS
LIN {X 36.6478,Y 11.0366,Z 62,A 8.9086,B 24.839,C -2.927,E1 25.1537,E2 -645.7747} C_DIS
LIN {X 37.2422,Y 8.825,Z 62,A 5.3578,B 24.8404,C -2.9148,E1 25.1561,E2 -642.2156} C_DIS
LIN {X 37.7903,Y 6.0625,Z 62,A 1.6598,B 24.8409,C -2.9102,E1 25.158,E2 -638.5283} C_DIS
LIN {X 37.9969,Y 4.5929,Z 62,A -0.543,B 24.8416,C -2.9036,E1 25.1588,E2 -636.323} C_DIS
LIN {X 38.1441,Y 3.1432,Z 62,A -3.2542,B 24.8432,C -2.8885,E1 25.1595,E2 -633.592} C_DIS
LIN {X 38.2709,Y 0.4491,Z 62,A -6.6123,B 24.8434,C -2.8866,E1 25.1598,E2 -630.2496} C_DIS
LIN {X 38.2492,Y -1.3711,Z 62,A -9.7969,B 24.8452,C -2.8708,E1 25.1596,E2 -627.0463} C_DIS
LIN {X 38.1207,Y -3.4151,Z 62,A -12.5246,B 24.8456,C -2.8665,E1 25.159,E2 -624.3247} C_DIS
LIN {X 37.868,Y -5.5548,Z 62,A -16.0131,B 24.8472,C -2.8522,E1 25.1577,E2 -620.823} C_DIS
LIN {X 37.3373,Y -8.4106,Z 62,A -20.8637,B 24.8495,C -2.8308,E1 25.155,E2 -615.9499} C_DIS
LIN {X 36.7293,Y -10.7619,Z 62,A -23.9295,B 24.8497,C -2.8286,E1 25.1527,E2 -612.8965} C_DIS
LIN {X 36.0087,Y -12.9707,Z 62,A -27.3966,B 24.8508,C -2.8182,E1 25.1495,E2 -609.4243} C_DIS
LIN {X 35.274,Y -14.8523,Z 62,A -29.974,B 24.851,C -2.8162,E1 25.1468,E2 -606.8565} C_DIS
LIN {X 34.493,Y -16.5854,Z 62,A -33.1274,B 24.8524,C -2.803,E1 25.1431,E2 -603.6889} C_DIS
LIN {X 33.5427,Y -18.4321,Z 62,A -36.2627,B 24.8534,C -2.7937,E1 25.139,E2 -600.548} C_DIS
LIN {X 32.3842,Y -20.3991,Z 62,A -39.9506,B 24.8548,C -2.7799,E1 25.1336,E2 -596.8464} C_DIS
LIN {X 30.7789,Y -22.7493,Z 62,A -43.7118,B 24.8552,C -2.7762,E1 25.1275,E2 -593.0947} C_DIS
LIN {X 29.6743,Y -24.172,Z 62,A -46.2451,B 24.8557,C -2.7718,E1 25.1232,E2 -590.5627} C_DIS
LIN {X 28.7927,Y -25.2156,Z 62,A -48.6975,B 24.8569,C -2.7604,E1 25.1186,E2 -588.0944} C_DIS
LIN {X 27.0386,Y -27.0874,Z 62,A -52.388,B 24.8576,C -2.7534,E1 25.1115,E2 -584.4032} C_DIS
LIN {X 25.4641,Y -28.5728,Z 62,A -55.7463,B 24.8586,C -2.7442,E1 25.1046,E2 -581.0368} C_DIS
LIN {X 23.5283,Y -30.1874,Z 62,A -59.1024,B 24.8588,C -2.7423,E1 25.0973,E2 -577.689} C_DIS
LIN {X 22.4018,Y -31.0328,Z 62,A -61.3281,B 24.8594,C -2.7363,E1 25.0923,E2 -575.4569} C_DIS
LIN {X 21.0009,Y -31.9971,Z 62,A -64.1117,B 24.8602,C -2.7279,E1 25.0858,E2 -572.6626} C_DIS
LIN {X 18.7839,Y -33.3464,Z 62,A -67.5903,B 24.8603,C -2.7269,E1 25.0775,E2 -569.1923} C_DIS
LIN {X 17.2735,Y -34.154,Z 62,A -70.6356,B 24.8615,C -2.7157,E1 25.0699,E2 -566.1289} C_DIS
LIN {X 15.6976,Y -34.906,Z 62,A -73.1533,B 24.8618,C -2.7131,E1 25.0635,E2 -563.6115} C_DIS
LIN {X 13.3113,Y -35.8845,Z 62,A -76.7824,B 24.862,C -2.7112,E1 25.054,E2 -559.9858} C_DIS
LIN {X 11.7403,Y -36.4282,Z 62,A -79.0576,B 24.862,C -2.7112,E1 25.048,E2 -557.7149} C_DIS
LIN {X 10.0144,Y -36.9399,Z 62,A -82.1081,B 24.8628,C -2.7033,E1 25.0398,E2 -554.6509} C_DIS
LIN {X 7.8882,Y -37.4512,Z 62,A -85.7505,B 24.8636,C -2.6953,E1 25.0298,E2 -550.9944} C_DIS
LIN {X 4.7975,Y -37.9716,Z 62,A -90.3592,B 24.8638,C -2.6933,E1 25.0171,E2 -546.385} C_DIS
LIN {X 1.4871,Y -38.2446,Z 62,A -94.8299,B 24.8633,C -2.6977,E1 25.0047,E2 -541.9269} C_DIS
LIN {X 0.2101,Y -38.2717,Z 62,A -95.9462,B 24.8623,C -2.7077,E1 25.0016,E2 -540.8345} C_DIS
Enddeposition()
LIN {X 0.2101,Y -38.2717,Z 62,A -95.9462,B 24.8623,C -2.7077,E1 25.0016,E2 -540.8345} C_DIS
Startdeposition()
$VEL.CP = VEL_PRINT
LIN {X 0.3798,Y -37.292,Z 62,A -94.1049,B 24.8584,C -2.7454,E1 25.007,E2 -542.765} C_DIS
LIN {X 4.6158,Y -37.0073,Z 62,A -88.4752,B 24.8593,C -2.7367,E1 25.0226,E2 -548.3708} C_DIS
LIN {X 7.0238,Y -36.6261,Z 62,A -84.9818,B 24.8593,C -2.7361,E1 25.0322,E2 -551.8592} C_DIS
LIN {X 8.6659,Y -36.2732,Z 62,A -81.6254,B 24.858,C -2.7492,E1 25.0414,E2 -555.242} C_DIS
LIN {X 12.594,Y -35.1033,Z 62,A -75.2736,B 24.8572,C -2.7575,E1 25.0583,E2 -561.6013} C_DIS
LIN {X 15.798,Y -33.7822,Z 62,A -70.7916,B 24.8576,C -2.7532,E1 25.0697,E2 -566.0622} C_DIS
LIN {X 17.4139,Y -32.9784,Z 62,A -67.9947,B 24.8571,C -2.758,E1 25.0766,E2 -568.863} C_DIS
LIN {X 19.0133,Y -32.0829,Z 62,A -65.1644,B 24.8566,C -2.7632,E1 25.0835,E2 -571.6971} C_DIS
LIN {X 20.6743,Y -31.039,Z 62,A -62.3816,B 24.8563,C -2.7655,E1 25.09,E2 -574.4762} C_DIS
LIN {X 21.7178,Y -30.3176,Z 62,A -60.2129,B 24.8556,C -2.7726,E1 25.095,E2 -576.6542} C_DIS
LIN {X 23.1933,Y -29.2044,Z 62,A -57.1249,B 24.8546,C -2.7823,E1 25.1018,E2 -579.7539} C_DIS
LIN {X 25.3351,Y -27.3673,Z 62,A -53.3687,B 24.8545,C -2.7833,E1 25.1097,E2 -583.4975} C_DIS
LIN {X 26.8633,Y -25.8685,Z 62,A -49.5005,B 24.8527,C -2.8,E1 25.1173,E2 -587.3887} C_DIS
LIN {X 28.3684,Y -24.2084,Z 62,A -46.3904,B 24.8524,C -2.8035,E1 25.123,E2 -590.4931} C_DIS
LIN {X 29.4078,Y -22.9356,Z 62,A -44.034,B 24.8519,C -2.8074,E1 25.1271,E2 -592.8479} C_DIS
LIN {X 30.4668,Y -21.5087,Z 62,A -41.0429,B 24.8507,C -2.8187,E1 25.132,E2 -595.8513} C_DIS
LIN {X 31.4827,Y -19.9922,Z 62,A -38.5107,B 24.8504,C -2.8222,E1 25.1359,E2 -598.3791} C_DIS
LIN {X 32.4337,Y -18.4094,Z 62,A -35.3939,B 24.8491,C -2.8346,E1 25.1403,E2 -601.509} C_DIS
LIN {X 33.513,Y -16.3612,Z 62,A -31.43,B 24.8473,C -2.8513,E1 25.1453,E2 -605.4915} C_DIS
LIN {X 34.7775,Y -13.4648,Z 62,A -26.7705,B 24.846,C -2.8627,E1 25.1502,E2 -610.1522} C_DIS
LIN {X 35.7679,Y -10.5583,Z 62,A -22.3655,B 24.845,C -2.8721,E1 25.154,E2 -614.5545} C_DIS
LIN {X 36.4434,Y -7.9174,Z 62,A -18.0335,B 24.8434,C -2.8873,E1 25.1568,E2 -618.8975} C_DIS
LIN {X 36.9555,Y -5.0093,Z 62,A -13.2669,B 24.8414,C -2.9052,E1 25.1588,E2 -623.6783} C_DIS
LIN {X 37.1857,Y -2.8388,Z 62,A -10.3802,B 24.8411,C -2.9082,E1 25.1595,E2 -626.5551} C_DIS
LIN {X 37.2777,Y -1.0841,Z 62,A -7.8149,B 24.8404,C -2.9146,E1 25.1598,E2 -629.1202} C_DIS
LIN {X 37.2812,Y 0.9781,Z 62,A -4.7509,B 24.8395,C -2.9228,E1 25.1597,E2 -632.1855} C_DIS
LIN {X 37.1828,Y 2.8744,Z 62,A -1.7044,B 24.8382,C -2.934,E1 25.1591,E2 -635.2403} C_DIS
LIN {X 37.0347,Y 4.3876,Z 62,A 0.5729,B 24.8375,C -2.9402,E1 25.1584,E2 -637.519} C_DIS
LIN {X 36.7615,Y 6.2787,Z 62,A 3.3871,B 24.8368,C -2.9473,E1 25.1572,E2 -640.3334} C_DIS
LIN {X 36.4215,Y 8.0184,Z 62,A 6.0852,B 24.8359,C -2.9551,E1 25.1556,E2 -643.0343} C_DIS
LIN {X 36.0127,Y 9.6904,Z 62,A 8.8571,B 24.8348,C -2.965,E1 25.1537,E2 -645.8135} C_DIS
LIN {X 35.3353,Y 11.9259,Z 62,A 11.9834,B 24.8344,C -2.9683,E1 25.1511,E2 -648.9298} C_DIS
LIN {X 34.7184,Y 13.6178,Z 62,A 15.5018,B 24.8322,C -2.9879,E1 25.1476,E2 -652.475} C_DIS
LIN {X 33.9409,Y 15.4548,Z 62,A 18.3781,B 24.8316,C -2.9935,E1 25.1443,E2 -655.3489} C_DIS
LIN {X 32.9506,Y 17.4665,Z 62,A 21.3677,B 24.8313,C -2.9957,E1 25.1405,E2 -658.328} C_DIS
LIN {X 32.0447,Y 19.0778,Z 62,A 24.9274,B 24.8292,C -3.0142,E1 25.1355,E2 -661.913} C_DIS
LIN {X 30.2317,Y 21.8379,Z 62,A 29.0163,B 24.8295,C -3.0118,E1 25.1291,E2 -665.9761} C_DIS
LIN {X 29.2193,Y 23.1743,Z 62,A 32.0027,B 24.8281,C -3.024,E1 25.124,E2 -668.9773} C_DIS
LIN {X 28.0065,Y 24.6265,Z 62,A 34.9807,B 24.8272,C -3.0316,E1 25.1185,E2 -671.9597} C_DIS
LIN {X 26.4595,Y 26.281,Z 62,A 38.0284,B 24.8272,C -3.0326,E1 25.1127,E2 -674.9966} C_DIS
LIN {X 25.54,Y 27.1758,Z 62,A 40.0717,B 24.8266,C -3.0376,E1 25.1086,E2 -677.0434} C_DIS
LIN {X 24.5311,Y 28.0896,Z 62,A 42.4592,B 24.8256,C -3.0459,E1 25.1035,E2 -679.4412} C_DIS
LIN {X 22.8495,Y 29.4742,Z 62,A 45.5762,B 24.8253,C -3.0486,E1 25.0968,E2 -682.553} C_DIS
LIN {X 21.5399,Y 30.4443,Z 62,A 48.2007,B 24.8246,C -3.0546,E1 25.0908,E2 -685.1822} C_DIS
LIN {X 19.9154,Y 31.5311,Z 62,A 51.0911,B 24.8243,C -3.0576,E1 25.0841,E2 -688.0703} C_DIS
LIN {X 18.4079,Y 32.4346,Z 62,A 54.1033,B 24.8233,C -3.0658,E1 25.0768,E2 -691.0928} C_DIS
LIN {X 16.723,Y 33.3345,Z 62,A 57.337,B 24.8224,C -3.0736,E1 25.0687,E2 -694.3362} C_DIS
LIN {X 13.5419,Y 34.7482,Z 62,A 61.9729,B 24.8229,C -3.0694,E1 25.0568,E2 -698.9512} C_DIS
LIN {X 11.7651,Y 35.3894,Z 62,A 65.1194,B 24.8222,C -3.0751,E1 25.0485,E2 -702.105} C_DIS
LIN {X 10.127,Y 35.8923,Z 62,A 67.4825,B 24.8224,C -3.0734,E1 25.0422,E2 -704.4599} C_DIS
LIN {X 8.7284,Y 36.258,Z 62,A 69.7018,B 24.8223,C -3.0746,E1 25.0362,E2 -706.6788} C_DIS
LIN {X 6.8036,Y 36.6678,Z 62,A 73.2908,B 24.8213,C -3.0833,E1 25.0263,E2 -710.2841} C_DIS
LIN {X 3.704,Y 37.109,Z 62,A 77.9971,B 24.8213,C -3.0828,E1 25.0133,E2 -714.9857} C_DIS
LIN {X 1.7014,Y 37.2549,Z 62,A 80.622,B 24.822,C -3.077,E1 25.006,E2 -717.5957} C_DIS
LIN {X 0.1788,Y 37.2932,Z 62,A 83.0286,B 24.822,C -3.0775,E1 24.9993,E2 -720.0032} C_DIS
LIN {X -1.4391,Y 37.2662,Z 62,A 85.6197,B 24.8219,C -3.0781,E1 24.992,E2 -722.5961} C_DIS
LIN {X -3.2208,Y 37.1549,Z 62,A 88.3,B 24.8221,C -3.0762,E1 24.9846,E2 -725.2729} C_DIS
LIN {X -4.7006,Y 36.9958,Z 62,A 90.9394,B 24.8218,C -3.0791,E1 24.9773,E2 -727.9211} C_DIS
LIN {X -7.3438,Y 36.5638,Z 62,A 94.6045,B 24.8227,C -3.0707,E1 24.9672,E2 -731.57} C_DIS
LIN {X -8.6182,Y 36.2842,Z 62,A 97.0896,B 24.8223,C -3.0745,E1 24.9604,E2 -734.0674} C_DIS
LIN {X -11.3372,Y 35.5289,Z 62,A 101.6603,B 24.8225,C -3.0726,E1 24.9482,E2 -738.6411} C_DIS
LIN {X -14.0073,Y 34.563,Z 62,A 105.3044,B 24.8241,C -3.0588,E1 24.9388,E2 -742.26} C_DIS
LIN {X -15.2664,Y 34.0258,Z 62,A 108.3324,B 24.8233,C -3.0661,E1 24.931,E2 -745.3127} C_DIS
LIN {X -18.7335,Y 32.2474,Z 62,A 113.1602,B 24.8259,C -3.0436,E1 24.9192,E2 -750.1003} C_DIS
LIN {X -20.2622,Y 31.309,Z 62,A 116.6381,B 24.8256,C -3.0463,E1 24.9109,E2 -753.5955} C_DIS
LIN {X -21.8956,Y 30.1891,Z 62,A 119.4301,B 24.8266,C -3.0376,E1 24.9046,E2 -756.3765} C_DIS
LIN {X -23.2788,Y 29.1368,Z 62,A 122.8757,B 24.8263,C -3.0402,E1 24.897,E2 -759.841} C_DIS
LIN {X -26.088,Y 26.6507,Z 62,A 127.4979,B 24.8291,C -3.0154,E1 24.8875,E2 -764.4227} C_DIS
LIN {X -27.0902,Y 25.6308,Z 62,A 130.9619,B 24.8282,C -3.0231,E1 24.8808,E2 -767.9199} C_DIS
LIN {X -29.7505,Y 22.4885,Z 62,A 136.3747,B 24.8311,C -2.9977,E1 24.8713,E2 -773.2973} C_DIS
LIN {X -31.2987,Y 20.2788,Z 62,A 141.4518,B 24.8313,C -2.9957,E1 24.8634,E2 -778.3949} C_DIS
LIN {X -32.6151,Y 18.0853,Z 62,A 145.3681,B 24.8326,C -2.9845,E1 24.858,E2 -782.3049} C_DIS
LIN {X -34.2141,Y 14.8396,Z 62,A 150.186,B 24.8352,C -2.9611,E1 24.8523,E2 -787.093} C_DIS
LIN {X -34.8673,Y 13.2318,Z 62,A 153.1178,B 24.8358,C -2.9557,E1 24.8493,E2 -790.0283} C_DIS
LIN {X -35.6631,Y 10.9077,Z 62,A 156.5306,B 24.8375,C -2.9408,E1 24.8464,E2 -793.425} C_DIS
LIN {X -36.0278,Y 9.6325,Z 62,A 158.7866,B 24.8379,C -2.9366,E1 24.8447,E2 -795.6841} C_DIS
LIN {X -36.4997,Y 7.6557,Z 62,A 161.8114,B 24.8391,C -2.9261,E1 24.8429,E2 -798.7012} C_DIS
LIN {X -36.7922,Y 6.0953,Z 62,A 164.2581,B 24.8399,C -2.9185,E1 24.8417,E2 -801.1445} C_DIS
LIN {X -37.0722,Y 4.0622,Z 62,A 167.8433,B 24.8406,C -2.9128,E1 24.8404,E2 -804.7373} C_DIS
LIN {X -37.2406,Y 1.9888,Z 62,A 170.7718,B 24.842,C -2.9002,E1 24.8399,E2 -807.6533} C_DIS
LIN {X -37.2914,Y 0.4626,Z 62,A 173.2157,B 24.8427,C -2.8938,E1 24.8398,E2 -810.0966} C_DIS
LIN {X -37.2638,Y -1.4947,Z 62,A 176.2515,B 24.8436,C -2.8847,E1 24.84,E2 -813.1289} C_DIS
LIN {X -37.1229,Y -3.5673,Z 62,A 179.5008,B 24.8447,C -2.8753,E1 24.8408,E2 -816.3753} C_DIS
LIN {X -36.8969,Y -5.4278,Z 62,A -177.3425,B 24.8453,C -2.8692,E1 24.842,E2 -819.5361} C_DIS
LIN {X -36.3848,Y -8.1859,Z 62,A -173.5025,B 24.8472,C -2.8516,E1 24.8441,E2 -823.3567} C_DIS
LIN {X -35.757,Y -10.5948,Z 62,A -169.2177,B 24.848,C -2.8448,E1 24.8473,E2 -827.65} C_DIS
LIN {X -35.0687,Y -12.689,Z 62,A -166.1783,B 24.8494,C -2.8316,E1 24.85,E2 -830.6753} C_DIS
LIN {X -34.4553,Y -14.2706,Z 62,A -163.4053,B 24.85,C -2.8259,E1 24.8529,E2 -833.45} C_DIS
LIN {X -33.5874,Y -16.2081,Z 62,A -160.4423,B 24.8512,C -2.814,E1 24.8564,E2 -836.4007} C_DIS
LIN {X -32.9971,Y -17.3784,Z 62,A -158.0176,B 24.8514,C -2.8127,E1 24.8595,E2 -838.8352} C_DIS
LIN {X -31.8213,Y -19.4481,Z 62,A -154.4366,B 24.8525,C -2.8024,E1 24.8646,E2 -842.4104} C_DIS
LIN {X -30.7774,Y -21.0618,Z 62,A -151.5435,B 24.8533,C -2.7945,E1 24.869,E2 -845.2989} C_DIS
LIN {X -29.7935,Y -22.4313,Z 62,A -148.8503,B 24.8538,C -2.7894,E1 24.8735,E2 -847.9929} C_DIS
LIN {X -28.3139,Y -24.2723,Z 62,A -145.0679,B 24.8545,C -2.7827,E1 24.8802,E2 -851.7769} C_DIS
LIN {X -26.75,Y -25.9861,Z 62,A -141.4454,B 24.8553,C -2.7758,E1 24.8872,E2 -855.3985} C_DIS
LIN {X -25.0195,Y -27.6564,Z 62,A -137.9111,B 24.8562,C -2.7668,E1 24.8944,E2 -858.9257} C_DIS
LIN {X -23.2695,Y -29.1441,Z 62,A -134.1824,B 24.8567,C -2.7625,E1 24.9024,E2 -862.6584} C_DIS
LIN {X -21.6886,Y -30.3384,Z 62,A -131.4131,B 24.8575,C -2.7544,E1 24.9086,E2 -865.4182} C_DIS
LIN {X -20.5497,Y -31.1211,Z 62,A -129.3389,B 24.8579,C -2.7506,E1 24.9134,E2 -867.4901} C_DIS
LIN {X -19.296,Y -31.9137,Z 62,A -126.5636,B 24.8577,C -2.7529,E1 24.9201,E2 -870.2796} C_DIS
LIN {X -16.6111,Y -33.3899,Z 62,A -122.4761,B 24.859,C -2.7398,E1 24.9301,E2 -874.3472} C_DIS
LIN {X -15.4577,Y -33.9393,Z 62,A -120.2457,B 24.859,C -2.7407,E1 24.9358,E2 -876.5854} C_DIS
LIN {X -13.75,Y -34.6665,Z 62,A -117.6067,B 24.8595,C -2.7354,E1 24.9426,E2 -879.2177} C_DIS
LIN {X -12.5138,Y -35.1315,Z 62,A -115.5054,B 24.8595,C -2.7345,E1 24.9481,E2 -881.3211} C_DIS
LIN {X -11.0993,Y -35.6037,Z 62,A -112.8845,B 24.8593,C -2.7368,E1 24.9551,E2 -883.952} C_DIS
LIN {X -8.6511,Y -36.2768,Z 62,A -109.158,B 24.8598,C -2.7325,E1 24.9652,E2 -887.6737} C_DIS
LIN {X -6.5504,Y -36.7139,Z 62,A -105.7934,B 24.8598,C -2.7321,E1 24.9744,E2 -891.0411} C_DIS
LIN {X -4.6911,Y -36.9975,Z 62,A -103.0272,B 24.86,C -2.7299,E1 24.982,E2 -893.8044} C_DIS
LIN {X -3.1676,Y -37.1594,Z 62,A -100.8141,B 24.8602,C -2.728,E1 24.9882,E2 -896.014} C_DIS
LIN {X -1.2338,Y -37.273,Z 62,A -97.1604,B 24.8593,C -2.737,E1 24.9984,E2 -899.69} C_DIS
LIN {X -1.2338,Y -37.273,Z 62,A -97.1604,B 24.8593,C -2.737,E1 24.9984,E2 -899.69} C_DIS
Enddeposition()
LIN {X 0.2259,Y -36.313,Z 62,A -96.7285,B 24.8599,C -2.7312,E1 24.9996,E2 -900.1081} C_DIS
Startdeposition()
$VEL.CP = VEL_PRINT
LIN {X -1.5145,Y -36.2824,Z 62,A -99.5448,B 24.86,C -2.73,E1 24.9917,E2 -897.2885} C_DIS
LIN {X -3.1836,Y -36.1745,Z 62,A -102.1919,B 24.86,C -2.73,E1 24.9844,E2 -894.6401} C_DIS
LIN {X -4.688,Y -36.0101,Z 62,A -104.3421,B 24.8597,C -2.7331,E1 24.9784,E2 -892.4961} C_DIS
LIN {X -6.507,Y -35.7263,Z 62,A -107.8438,B 24.8603,C -2.7269,E1 24.9687,E2 -888.9764} C_DIS
LIN {X -8.9633,Y -35.1903,Z 62,A -111.5567,B 24.8598,C -2.7318,E1 24.9586,E2 -885.2702} C_DIS
LIN {X -10.8933,Y -34.6419,Z 62,A -114.6519,B 24.8595,C -2.7348,E1 24.9504,E2 -882.1768} C_DIS
LIN {X -13.595,Y -33.6733,Z 62,A -119.3328,B 24.8593,C -2.7371,E1 24.9381,E2 -877.4917} C_DIS
LIN {X -15.3047,Y -32.9313,Z 62,A -122.1053,B 24.8588,C -2.7421,E1 24.9311,E2 -874.7244} C_DIS
LIN {X -16.8467,Y -32.1698,Z 62,A -124.9012,B 24.8585,C -2.7445,E1 24.9241,E2 -871.9267} C_DIS
LIN {X -18.5754,Y -31.2037,Z 62,A -128.054,B 24.8581,C -2.7485,E1 24.9165,E2 -868.774} C_DIS
LIN {X -20.4782,Y -29.9895,Z 62,A -131.4375,B 24.8574,C -2.7558,E1 24.9086,E2 -865.3969} C_DIS
LIN {X -21.575,Y -29.2104,Z 62,A -134.1896,B 24.8577,C -2.7528,E1 24.9024,E2 -862.6281} C_DIS
LIN {X -24.0635,Y -27.1974,Z 62,A -138.6999,B 24.8561,C -2.7676,E1 24.8927,E2 -858.1358} C_DIS
LIN {X -25.856,Y -25.4978,Z 62,A -143.0514,B 24.8558,C -2.771,E1 24.884,E2 -853.7741} C_DIS
LIN {X -27.8087,Y -23.3524,Z 62,A -147.9687,B 24.8551,C -2.7778,E1 24.875,E2 -848.851} C_DIS
LIN {X -29.8611,Y -20.6646,Z 62,A -152.7163,B 24.8531,C -2.7962,E1 24.8672,E2 -844.1243} C_DIS
LIN {X -30.7668,Y -19.2901,Z 62,A -155.0523,B 24.8522,C -2.8052,E1 24.8637,E2 -841.7981} C_DIS
LIN {X -31.6029,Y -17.8886,Z 62,A -157.9082,B 24.8518,C -2.8092,E1 24.8596,E2 -838.937} C_DIS
LIN {X -32.4495,Y -16.3022,Z 62,A -160.72,B 24.8509,C -2.817,E1 24.856,E2 -836.1289} C_DIS
LIN {X -33.2834,Y -14.5231,Z 62,A -164.2246,B 24.8504,C -2.8219,E1 24.852,E2 -832.6166} C_DIS
LIN {X -34.2983,Y -11.9308,Z 62,A -168.0261,B 24.8485,C -2.8398,E1 24.8483,E2 -828.8366} C_DIS
LIN {X -34.6918,Y -10.7323,Z 62,A -170.5019,B 24.8483,C -2.8412,E1 24.8462,E2 -826.35} C_DIS
LIN {X -35.422,Y -8.0011,Z 62,A -175.2833,B 24.8472,C -2.8517,E1 24.843,E2 -821.5656} C_DIS
LIN {X -35.9337,Y -5.2429,Z 62,A -179.065,B 24.8451,C -2.8709,E1 24.8413,E2 -817.8074} C_DIS
LIN {X -36.1175,Y -3.7714,Z 62,A 178.0448,B 24.8449,C -2.8732,E1 24.8404,E2 -814.9055} C_DIS
LIN {X -36.2743,Y -1.7026,Z 62,A 175.1574,B 24.8434,C -2.8868,E1 24.8399,E2 -812.0332} C_DIS
LIN {X -36.3143,Y 0.0076,Z 62,A 172.3134,B 24.8426,C -2.8939,E1 24.8398,E2 -809.1892} C_DIS
LIN {X -36.2672,Y 1.8483,Z 62,A 169.6266,B 24.8414,C -2.905,E1 24.8401,E2 -806.5126} C_DIS
LIN {X -36.0426,Y 4.4294,Z 62,A 164.3098,B 24.8412,C -2.9071,E1 24.8417,E2 -801.169} C_DIS
LIN {X -35.6411,Y 6.9587,Z 62,A 160.394,B 24.8397,C -2.9207,E1 24.8437,E2 -797.2627} C_DIS
LIN {X -34.6971,Y 10.7151,Z 62,A 155.158,B 24.8368,C -2.9471,E1 24.8475,E2 -792.0595} C_DIS
LIN {X -34.1203,Y 12.4303,Z 62,A 152.0186,B 24.8361,C -2.9532,E1 24.8504,E2 -788.9169} C_DIS
LIN {X -33.2306,Y 14.6436,Z 62,A 148.0572,B 24.8351,C -2.9626,E1 24.8547,E2 -784.9559} C_DIS
LIN {X -31.9074,Y 17.3385,Z 62,A 143.9688,B 24.8329,C -2.9821,E1 24.8599,E2 -780.8922} C_DIS
LIN {X -31.292,Y 18.426,Z 62,A 141.218,B 24.833,C -2.9805,E1 24.8638,E2 -778.1235} C_DIS
LIN {X -29.5922,Y 21.0478,Z 62,A 136.9654,B 24.8308,C -3.0001,E1 24.8703,E2 -773.8964} C_DIS
LIN {X -28.8062,Y 22.1113,Z 62,A 133.8314,B 24.8313,C -2.9958,E1 24.8757,E2 -770.7373} C_DIS
LIN {X -26.1557,Y 25.1909,Z 62,A 128.3992,B 24.8285,C -3.0208,E1 24.8857,E2 -765.3406} C_DIS
LIN {X -24.1569,Y 27.1138,Z 62,A 122.9157,B 24.8285,C -3.0201,E1 24.897,E2 -759.8332} C_DIS
LIN {X -21.7781,Y 29.0587,Z 62,A 118.2831,B 24.8272,C -3.0322,E1 24.9072,E2 -755.2126} C_DIS
LIN {X -18.883,Y 31.0183,Z 62,A 113.3103,B 24.8254,C -3.048,E1 24.9188,E2 -750.2612} C_DIS
LIN {X -16.5144,Y 32.3416,Z 62,A 108.5765,B 24.8251,C -3.0504,E1 24.9305,E2 -745.52} C_DIS
LIN {X -14.192,Y 33.4261,Z 62,A 104.9283,B 24.8239,C -3.0604,E1 24.9397,E2 -741.8867} C_DIS
LIN {X -12.2071,Y 34.2013,Z 62,A 101.481,B 24.8235,C -3.0637,E1 24.9487,E2 -738.4404} C_DIS
LIN {X -10.2433,Y 34.8394,Z 62,A 98.2949,B 24.823,C -3.0681,E1 24.9572,E2 -735.2592} C_DIS
LIN {X -8.5749,Y 35.2871,Z 62,A 95.7194,B 24.8225,C -3.0724,E1 24.9642,E2 -732.6902} C_DIS
LIN {X -7.1623,Y 35.6009,Z 62,A 93.5063,B 24.8222,C -3.0751,E1 24.9702,E2 -730.4808} C_DIS
LIN {X -5.8849,Y 35.8338,Z 62,A 90.9214,B 24.8228,C -3.0705,E1 24.9774,E2 -727.8826} C_DIS
LIN {X -3.0398,Y 36.1868,Z 62,A 86.882,B 24.8218,C -3.0784,E1 24.9885,E2 -723.8595} C_DIS
LIN {X -1.3484,Y 36.2893,Z 62,A 84.3466,B 24.8215,C -3.0809,E1 24.9956,E2 -721.3296} C_DIS
LIN {X 0.226,Y 36.3133,Z 62,A 81.6004,B 24.8218,C -3.0784,E1 25.0033,E2 -718.5773} C_DIS
LIN {X 2.2009,Y 36.2477,Z 62,A 78.354,B 24.822,C -3.077,E1 25.0123,E2 -715.3286} C_DIS
LIN {X 4.399,Y 36.0463,Z 62,A 75.1943,B 24.8216,C -3.0805,E1 25.0211,E2 -712.1792} C_DIS
LIN {X 6.3247,Y 35.7591,Z 62,A 72.0985,B 24.8217,C -3.0792,E1 25.0296,E2 -709.0835} C_DIS
LIN {X 8.2509,Y 35.3643,Z 62,A 69.2359,B 24.8216,C -3.0808,E1 25.0374,E2 -706.2283} C_DIS
LIN {X 9.5766,Y 35.0286,Z 62,A 66.4695,B 24.8226,C -3.0718,E1 25.0449,E2 -703.4449} C_DIS
LIN {X 12.4788,Y 34.1026,Z 62,A 62.0854,B 24.8224,C -3.0734,E1 25.0565,E2 -699.0729} C_DIS
LIN {X 13.7626,Y 33.6051,Z 62,A 59.4958,B 24.8233,C -3.0658,E1 25.0632,E2 -696.4712} C_DIS
LIN {X 15.9846,Y 32.6069,Z 62,A 56.1006,B 24.8231,C -3.0673,E1 25.0718,E2 -693.0882} C_DIS
LIN {X 17.1879,Y 31.989,Z 62,A 53.9025,B 24.8235,C -3.0637,E1 25.0773,E2 -690.8877} C_DIS
LIN {X 18.5719,Y 31.2056,Z 62,A 51.4061,B 24.8239,C -3.0604,E1 25.0833,E2 -688.391} C_DIS
LIN {X 20.2486,Y 30.1449,Z 62,A 47.855,B 24.8251,C -3.0499,E1 25.0916,E2 -684.8265} C_DIS
LIN {X 22.1451,Y 28.7802,Z 62,A 44.6484,B 24.8251,C -3.0502,E1 25.0988,E2 -681.6322} C_DIS
LIN {X 23.2341,Y 27.9083,Z 62,A 42.1716,B 24.826,C -3.0423,E1 25.1042,E2 -679.1462} C_DIS
LIN {X 24.8421,Y 26.4873,Z 62,A 38.857,B 24.8267,C -3.0367,E1 25.111,E2 -675.8315} C_DIS
LIN {X 26.2732,Y 25.0681,Z 62,A 35.8895,B 24.8271,C -3.0331,E1 25.1168,E2 -672.8681} C_DIS
LIN {X 27.3075,Y 23.9377,Z 62,A 33.568,B 24.8275,C -3.0291,E1 25.1212,E2 -670.5476} C_DIS
LIN {X 28.1296,Y 22.9655,Z 62,A 30.9317,B 24.8291,C -3.0156,E1 25.1259,E2 -667.8914} C_DIS
LIN {X 29.5252,Y 21.1417,Z 62,A 27.3467,B 24.83,C -3.0074,E1 25.1318,E2 -664.3042} C_DIS
LIN {X 31.0967,Y 18.754,Z 62,A 23.3509,B 24.8304,C -3.0035,E1 25.1378,E2 -660.3192} C_DIS
LIN {X 32.3011,Y 16.5936,Z 62,A 18.5393,B 24.8331,C -2.9798,E1 25.1441,E2 -655.4768} C_DIS
LIN {X 33.7743,Y 13.3419,Z 62,A 13.5609,B 24.8338,C -2.9737,E1 25.1496,E2 -650.5113} C_DIS
LIN {X 34.5565,Y 11.1605,Z 62,A 10.1503,B 24.8346,C -2.9668,E1 25.1527,E2 -647.1036} C_DIS
LIN {X 35.0479,Y 9.5052,Z 62,A 7.2878,B 24.8357,C -2.9567,E1 25.1548,E2 -644.2335} C_DIS
LIN {X 35.5924,Y 7.2036,Z 62,A 3.8721,B 24.8364,C -2.9502,E1 25.1569,E2 -640.8223} C_DIS
LIN {X 35.8634,Y 5.7013,Z 62,A 1.2832,B 24.8376,C -2.9401,E1 25.1581,E2 -638.2248} C_DIS
LIN {X 36.1144,Y 3.8016,Z 62,A -1.6037,B 24.8384,C -2.9329,E1 25.1591,E2 -635.3378} C_DIS
LIN {X 36.2546,Y 2.0764,Z 62,A -4.1491,B 24.839,C -2.9272,E1 25.1596,E2 -632.794} C_DIS
LIN {X 36.3048,Y 0.8342,Z 62,A -6.6619,B 24.8406,C -2.9127,E1 25.1598,E2 -630.2618} C_DIS
LIN {X 36.2452,Y -2.244,Z 62,A -12.166,B 24.8433,C -2.8877,E1 25.1591,E2 -624.7313} C_DIS
LIN {X 35.7559,Y -6.3428,Z 62,A -17.7492,B 24.844,C -2.8814,E1 25.1569,E2 -619.1661} C_DIS
LIN {X 35.2811,Y -8.5989,Z 62,A -21.233,B 24.845,C -2.8725,E1 25.1548,E2 -615.6814} C_DIS
LIN {X 34.8064,Y -10.3546,Z 62,A -24.5737,B 24.8467,C -2.8565,E1 25.1522,E2 -612.322} C_DIS
LIN {X 33.7265,Y -13.4633,Z 62,A -29.2077,B 24.8475,C -2.8493,E1 25.1477,E2 -607.6968} C_DIS
LIN {X 32.9567,Y -15.2487,Z 62,A -32.5766,B 24.8489,C -2.8357,E1 25.1439,E2 -604.3142} C_DIS
LIN {X 31.7642,Y -17.5998,Z 62,A -36.633,B 24.85,C -2.8253,E1 25.1386,E2 -600.2545} C_DIS
LIN {X 30.4664,Y -19.7619,Z 62,A -40.6702,B 24.8513,C -2.8134,E1 25.1326,E2 -596.2095} C_DIS
LIN {X 29.3366,Y -21.4027,Z 62,A -43.395,B 24.8515,C -2.8112,E1 25.1282,E2 -593.4928} C_DIS
LIN {X 28.2789,Y -22.782,Z 62,A -46.3899,B 24.8527,C -2.8003,E1 25.123,E2 -590.4862} C_DIS
LIN {X 26.8003,Y -24.5041,Z 62,A -49.9148,B 24.8535,C -2.7922,E1 25.1165,E2 -586.9579} C_DIS
LIN {X 25.4552,Y -25.8987,Z 62,A -52.7479,B 24.854,C -2.7882,E1 25.1109,E2 -584.1273} C_DIS
LIN {X 24.2459,Y -27.0341,Z 62,A -55.4302,B 24.8547,C -2.7813,E1 25.1054,E2 -581.4394} C_DIS
LIN {X 22.8571,Y -28.2181,Z 62,A -58.4415,B 24.8556,C -2.7731,E1 25.0989,E2 -578.4204} C_DIS
LIN {X 21.0337,Y -29.6023,Z 62,A -61.832,B 24.856,C -2.7689,E1 25.0913,E2 -575.032} C_DIS
LIN {X 19.7566,Y -30.4698,Z 62,A -64.1306,B 24.8563,C -2.7661,E1 25.086,E2 -572.7345} C_DIS
LIN {X 18.0192,Y -31.5281,Z 62,A -67.9326,B 24.8577,C -2.7522,E1 25.0768,E2 -568.911} C_DIS
LIN {X 16.0141,Y -32.5925,Z 62,A -71.0354,B 24.8577,C -2.7529,E1 25.0691,E2 -565.8184} C_DIS
LIN {X 14.5705,Y -33.2621,Z 62,A -73.6764,B 24.8582,C -2.7474,E1 25.0623,E2 -563.171} C_DIS
LIN {X 12.4585,Y -34.11,Z 62,A -76.9664,B 24.8583,C -2.7466,E1 25.0538,E2 -559.8863} C_DIS
LIN {X 11.0737,Y -34.5845,Z 62,A -79.2949,B 24.8586,C -2.7436,E1 25.0476,E2 -557.5551} C_DIS
LIN {X 9.4245,Y -35.0697,Z 62,A -82.2025,B 24.8592,C -2.7381,E1 25.0398,E2 -554.6393} C_DIS
LIN {X 7.3335,Y -35.5658,Z 62,A -85.7943,B 24.8598,C -2.7324,E1 25.03,E2 -551.0388} C_DIS
LIN {X 5.2774,Y -35.9289,Z 62,A -88.7814,B 24.8596,C -2.734,E1 25.0217,E2 -548.0584} C_DIS
LIN {X 2.9609,Y -36.1931,Z 62,A -93.0264,B 24.8606,C -2.7249,E1 25.0099,E2 -543.7943} C_DIS
LIN {X 0.2259,Y -36.313,Z 62,A -96.7284,B 24.8599,C -2.7312,E1 24.9996,E2 -540.1081} C_DIS
Enddeposition()
LIN {X 0.2259,Y -36.313,Z 62,A -96.7284,B 24.8599,C -2.7312,E1 24.9996,E2 -540.1081} C_DIS
Startdeposition()
$VEL.CP = VEL_PRINT
LIN {X 1.2682,Y -35.312,Z 62,A -93.5151,B 24.8561,C -2.7675,E1 25.0088,E2 -543.4072} C_DIS
LIN {X 3.3153,Y -35.1785,Z 62,A -90.4229,B 24.8563,C -2.7661,E1 25.0174,E2 -546.4945} C_DIS
LIN {X 5.258,Y -34.9404,Z 62,A -86.927,B 24.8556,C -2.7723,E1 25.0271,E2 -550.0021} C_DIS
LIN {X 8.1824,Y -34.3744,Z 62,A -81.8634,B 24.8549,C -2.7796,E1 25.0409,E2 -555.0765} C_DIS
LIN {X 11.0176,Y -33.573,Z 62,A -77.8325,B 24.8553,C -2.7751,E1 25.0517,E2 -559.0896} C_DIS
LIN {X 12.2849,Y -33.1302,Z 62,A -74.7064,B 24.8537,C -2.7907,E1 25.0599,E2 -562.2461} C_DIS
LIN {X 16.1341,Y -31.4358,Z 62,A -68.7935,B 24.8539,C -2.7886,E1 25.0749,E2 -568.1391} C_DIS
LIN {X 18.1492,Y -30.3176,Z 62,A -64.4351,B 24.8523,C -2.8039,E1 25.0855,E2 -572.5204} C_DIS
LIN {X 20.3496,Y -28.8869,Z 62,A -60.7598,B 24.8523,C -2.8039,E1 25.0939,E2 -576.1835} C_DIS
LIN {X 21.6446,Y -27.9289,Z 62,A -58.246,B 24.8519,C -2.808,E1 25.0995,E2 -578.6977} C_DIS
LIN {X 22.8521,Y -26.9498,Z 62,A -55.6388,B 24.8512,C -2.8147,E1 25.1051,E2 -581.3109} C_DIS
LIN {X 24.1972,Y -25.749,Z 62,A -52.7154,B 24.8505,C -2.8214,E1 25.1112,E2 -584.2382} C_DIS
LIN {X 25.5488,Y -24.4088,Z 62,A -49.8823,B 24.8501,C -2.8251,E1 25.1167,E2 -587.0681} C_DIS
LIN {X 26.3848,Y -23.5024,Z 62,A -47.692,B 24.8492,C -2.8328,E1 25.1208,E2 -589.2669} C_DIS
LIN {X 27.5812,Y -22.087,Z 62,A -44.6244,B 24.8483,C -2.8414,E1 25.1263,E2 -592.3407} C_DIS
LIN {X 28.3877,Y -21.0383,Z 62,A -41.8996,B 24.8468,C -2.8557,E1 25.1308,E2 -595.0863} C_DIS
LIN {X 30.5253,Y -17.7979,Z 62,A -36.58,B 24.8465,C -2.8585,E1 25.1388,E2 -600.3858} C_DIS
LIN {X 31.598,Y -15.8145,Z 62,A -31.8568,B 24.8436,C -2.885,E1 25.1449,E2 -605.1468} C_DIS
LIN {X 32.7781,Y -13.1946,Z 62,A -28.0348,B 24.8435,C -2.8862,E1 25.149,E2 -608.9506} C_DIS
LIN {X 33.433,Y -11.4335,Z 62,A -25.2225,B 24.8429,C -2.8919,E1 25.1517,E2 -611.7605} C_DIS
LIN {X 33.845,Y -10.151,Z 62,A -22.5625,B 24.8413,C -2.9057,E1 25.1539,E2 -614.4383} C_DIS
LIN {X 34.4799,Y -7.725,Z 62,A -18.8752,B 24.8406,C -2.9125,E1 25.1563,E2 -618.1204} C_DIS
LIN {X 34.797,Y -6.1397,Z 62,A -15.7441,B 24.8388,C -2.9285,E1 25.1579,E2 -621.2708} C_DIS
LIN {X 35.1952,Y -3.1276,Z 62,A -11.665,B 24.8386,C -2.931,E1 25.1592,E2 -625.3319} C_DIS
LIN {X 35.2789,Y -1.9779,Z 62,A -9.5541,B 24.8375,C -2.9406,E1 25.1596,E2 -627.4527} C_DIS
LIN {X 35.3337,Y -0.2209,Z 62,A -6.6131,B 24.8364,C -2.9509,E1 25.1598,E2 -630.4007} C_DIS
LIN {X 35.3037,Y 1.4724,Z 62,A -3.9725,B 24.8356,C -2.9578,E1 25.1595,E2 -633.042} C_DIS
LIN {X 35.2076,Y 2.9936,Z 62,A -1.601,B 24.8349,C -2.964,E1 25.1591,E2 -635.4141} C_DIS
LIN {X 34.9877,Y 4.9372,Z 62,A 2.3046,B 24.8326,C -2.9849,E1 25.1576,E2 -639.3461} C_DIS
LIN {X 34.6379,Y 6.9806,Z 62,A 5.3098,B 24.832,C -2.9897,E1 25.1561,E2 -642.3451} C_DIS
LIN {X 34.0832,Y 9.32,Z 62,A 9.091,B 24.8309,C -2.9995,E1 25.1534,E2 -646.1277} C_DIS
LIN {X 33.5155,Y 11.191,Z 62,A 12.0434,B 24.8302,C -3.0055,E1 25.1509,E2 -649.0776} C_DIS
LIN {X 32.944,Y 12.7755,Z 62,A 15.3086,B 24.8284,C -3.0213,E1 25.1477,E2 -652.3619} C_DIS
LIN {X 31.9114,Y 15.1723,Z 62,A 19.2768,B 24.8275,C -3.029,E1 25.1431,E2 -656.327} C_DIS
LIN {X 30.7637,Y 17.3819,Z 62,A 22.7893,B 24.8272,C -3.0321,E1 25.1385,E2 -659.8283} C_DIS
LIN {X 30.1474,Y 18.4297,Z 62,A 25.1988,B 24.8259,C -3.0435,E1 25.135,E2 -662.2525} C_DIS
LIN {X 28.8185,Y 20.4454,Z 62,A 28.9755,B 24.825,C -3.0512,E1 25.129,E2 -666.0288} C_DIS
LIN {X 27.637,Y 22.0165,Z 62,A 32.0725,B 24.8243,C -3.0573,E1 25.1237,E2 -669.1259} C_DIS
LIN {X 26.3263,Y 23.5677,Z 62,A 34.8658,B 24.8243,C -3.0576,E1 25.1186,E2 -671.9071} C_DIS
LIN {X 25.0628,Y 24.9068,Z 62,A 38.5533,B 24.8224,C -3.0738,E1 25.1114,E2 -675.6172} C_DIS
LIN {X 23.1366,Y 26.7059,Z 62,A 43.0696,B 24.821,C -3.0855,E1 25.102,E2 -680.143} C_DIS
LIN {X 21.0952,Y 28.3467,Z 62,A 47.3529,B 24.8201,C -3.0934,E1 25.0925,E2 -684.4294} C_DIS
LIN {X 18.4801,Y 30.1168,Z 62,A 51.6727,B 24.8204,C -3.0904,E1 25.0825,E2 -688.7281} C_DIS
LIN {X 17.3578,Y 30.7773,Z 62,A 53.8564,B 24.82,C -3.0943,E1 25.0772,E2 -690.9144} C_DIS
LIN {X 15.9419,Y 31.534,Z 62,A 56.4854,B 24.8196,C -3.098,E1 25.0707,E2 -693.5448} C_DIS
LIN {X 14.5728,Y 32.1893,Z 62,A 58.799,B 24.8195,C -3.0989,E1 25.0648,E2 -695.8546} C_DIS
LIN {X 12.8523,Y 32.9141,Z 62,A 62.2963,B 24.8184,C -3.1079,E1 25.0557,E2 -699.3655} C_DIS
LIN {X 11.0392,Y 33.566,Z 62,A 65.0271,B 24.8187,C -3.1055,E1 25.0486,E2 -702.0852} C_DIS
LIN {X 9.3911,Y 34.0636,Z 62,A 68.1251,B 24.818,C -3.1113,E1 25.0402,E2 -705.1916} C_DIS
LIN {X 7.3231,Y 34.5678,Z 62,A 71.7212,B 24.8176,C -3.1148,E1 25.0304,E2 -708.7911} C_DIS
LIN {X 4.9026,Y 34.9926,Z 62,A 75.1962,B 24.8182,C -3.1098,E1 25.0209,E2 -712.2508} C_DIS
LIN {X 3.4982,Y 35.161,Z 62,A 77.5331,B 24.8181,C -3.1106,E1 25.0144,E2 -714.5882} C_DIS
LIN {X 2.0334,Y 35.2759,Z 62,A 79.8529,B 24.8181,C -3.1099,E1 25.0079,E2 -716.9053} C_DIS
LIN {X 0.4926,Y 35.3312,Z 62,A 82.5036,B 24.818,C -3.1114,E1 25.0005,E2 -719.559} C_DIS
LIN {X -1.3857,Y 35.3073,Z 62,A 85.518,B 24.8181,C -3.1102,E1 24.9921,E2 -722.5709} C_DIS
LIN {X -2.8589,Y 35.2185,Z 62,A 88.7111,B 24.8172,C -3.1184,E1 24.9832,E2 -725.7848} C_DIS
LIN {X -6.6994,Y 34.6934,Z 62,A 93.9331,B 24.8191,C -3.1022,E1 24.9689,E2 -730.9728} C_DIS
LIN {X -9.2073,Y 34.1136,Z 62,A 99.2306,B 24.8181,C -3.1106,E1 24.9544,E2 -736.2978} C_DIS
LIN {X -11.7129,Y 33.3365,Z 62,A 102.6727,B 24.8197,C -3.0969,E1 24.9454,E2 -739.7136} C_DIS
LIN {X -13.7389,Y 32.5539,Z 62,A 106.5808,B 24.8197,C -3.0962,E1 24.9352,E2 -743.6287} C_DIS
LIN {X -16.0759,Y 31.4655,Z 62,A 110.8431,B 24.8204,C -3.0906,E1 24.9246,E2 -747.8887} C_DIS
LIN {X -17.9867,Y 30.4137,Z 62,A 113.9705,B 24.8216,C -3.0803,E1 24.917,E2 -751.0008} C_DIS
LIN {X -19.5991,Y 29.4009,Z 62,A 117.2485,B 24.8221,C -3.0765,E1 24.9093,E2 -754.2802} C_DIS
LIN {X -21.4516,Y 28.0779,Z 62,A 121.0929,B 24.8228,C -3.0706,E1 24.9007,E2 -758.1241} C_DIS
LIN {X -23.4689,Y 26.4148,Z 62,A 125.5344,B 24.8236,C -3.0633,E1 24.8913,E2 -762.5655} C_DIS
LIN {X -25.2491,Y 24.7189,Z 62,A 129.211,B 24.825,C -3.051,E1 24.884,E2 -766.2282} C_DIS
LIN {X -26.8751,Y 22.94,Z 62,A 133.3816,B 24.8258,C -3.0438,E1 24.8763,E2 -770.4003} C_DIS
LIN {X -28.5459,Y 20.8242,Z 62,A 137.8672,B 24.827,C -3.0335,E1 24.8687,E2 -774.8827} C_DIS
LIN {X -29.821,Y 18.9538,Z 62,A 141.0995,B 24.8286,C -3.0195,E1 24.8638,E2 -778.0976} C_DIS
LIN {X -30.7567,Y 17.3948,Z 62,A 144.1285,B 24.8295,C -3.012,E1 24.8596,E2 -781.1243} C_DIS
LIN {X -31.756,Y 15.4951,Z 62,A 147.8183,B 24.8304,C -3.0038,E1 24.8549,E2 -784.8145} C_DIS
LIN {X -32.8135,Y 13.107,Z 62,A 152.4225,B 24.8315,C -2.9946,E1 24.8499,E2 -789.4222} C_DIS
LIN {X -33.554,Y 11.0763,Z 62,A 155.1981,B 24.8334,C -2.9775,E1 24.8474,E2 -792.1727} C_DIS
LIN {X -34.1276,Y 9.1554,Z 62,A 159.072,B 24.8339,C -2.9731,E1 24.8445,E2 -796.0584} C_DIS
LIN {X -34.5747,Y 7.2849,Z 62,A 161.7796,B 24.8354,C -2.9598,E1 24.8428,E2 -798.7502} C_DIS
LIN {X -35.0069,Y 4.7973,Z 62,A 166.3044,B 24.8364,C -2.9509,E1 24.8409,E2 -803.2804} C_DIS
LIN {X -35.2566,Y 2.3429,Z 62,A 169.4971,B 24.8385,C -2.9313,E1 24.8401,E2 -806.4454} C_DIS
LIN {X -35.3322,Y 0.4226,Z 62,A 173.6141,B 24.8386,C -2.9303,E1 24.8398,E2 -810.5848} C_DIS
LIN {X -35.2647,Y -2.2226,Z 62,A 177.2925,B 24.8407,C -2.9115,E1 24.8402,E2 -814.2404} C_DIS
LIN {X -35.1133,Y -3.9496,Z 62,A -179.3162,B 24.8411,C -2.908,E1 24.8412,E2 -817.6436} C_DIS
LIN {X -34.585,Y -7.2393,Z 62,A -174.5294,B 24.8435,C -2.8861,E1 24.8435,E2 -822.4063} C_DIS
LIN {X -34.1478,Y -9.0789,Z 62,A -171.3803,B 24.8444,C -2.8777,E1 24.8456,E2 -825.5537} C_DIS
LIN {X -33.6196,Y -10.8736,Z 62,A -168.6634,B 24.8457,C -2.8659,E1 24.8478,E2 -828.2582} C_DIS
LIN {X -32.901,Y -12.8856,Z 62,A -163.7538,B 24.8453,C -2.8692,E1 24.8526,E2 -833.2034} C_DIS
LIN {X -31.5572,Y -15.8944,Z 62,A -159.2794,B 24.8478,C -2.8465,E1 24.8579,E2 -837.6478} C_DIS
LIN {X -30.7688,Y -17.3731,Z 62,A -156.634,B 24.8486,C -2.8387,E1 24.8615,E2 -840.2883} C_DIS
LIN {X -29.9935,Y -18.6791,Z 62,A -154.2187,B 24.8493,C -2.832,E1 24.865,E2 -842.6999} C_DIS
LIN {X -29.1957,Y -19.9031,Z 62,A -151.7563,B 24.8499,C -2.827,E1 24.8688,E2 -845.1626} C_DIS
LIN {X -28.1187,Y -21.3979,Z 62,A -148.0177,B 24.8499,C -2.8271,E1 24.8751,E2 -848.9196} C_DIS
LIN {X -26.1239,Y -23.7923,Z 62,A -143.1442,B 24.8512,C -2.8142,E1 24.884,E2 -853.7842} C_DIS
LIN {X -23.8347,Y -26.085,Z 62,A -138.5556,B 24.8531,C -2.7969,E1 24.8932,E2 -858.3506} C_DIS
LIN {X -22.0975,Y -27.5723,Z 62,A -134.0775,B 24.8529,C -2.798,E1 24.9028,E2 -862.8484} C_DIS
LIN {X -19.9931,Y -29.1348,Z 62,A -130.2213,B 24.8541,C -2.7869,E1 24.9116,E2 -866.6915} C_DIS
LIN {X -18.2246,Y -30.272,Z 62,A -126.894,B 24.8547,C -2.7811,E1 24.9195,E2 -870.0153} C_DIS
LIN {X -17.0864,Y -30.9283,Z 62,A -124.357,B 24.8546,C -2.7826,E1 24.9257,E2 -872.5634} C_DIS
LIN {X -14.5577,Y -32.1961,Z 62,A -120.408,B 24.8558,C -2.7703,E1 24.9356,E2 -876.4933} C_DIS
LIN {X -13.3467,Y -32.7167,Z 62,A -118.0208,B 24.8558,C -2.771,E1 24.9417,E2 -878.8874} C_DIS
LIN {X -11.5751,Y -33.3848,Z 62,A -114.9475,B 24.856,C -2.7684,E1 24.9498,E2 -881.9607} C_DIS
LIN {X -10.0708,Y -33.8688,Z 62,A -112.2482,B 24.856,C -2.7682,E1 24.957,E2 -884.6641} C_DIS
LIN {X -7.9938,Y -34.4182,Z 62,A -108.804,B 24.8563,C -2.7658,E1 24.9663,E2 -888.1076} C_DIS
LIN {X -6.072,Y -34.8092,Z 62,A -105.6894,B 24.8565,C -2.7639,E1 24.9749,E2 -891.2211} C_DIS
LIN {X -4.2103,Y -35.0827,Z 62,A -102.5918,B 24.8565,C -2.7639,E1 24.9835,E2 -894.3209} C_DIS
LIN {X -2.2175,Y -35.2651,Z 62,A -99.6594,B 24.8569,C -2.7601,E1 24.9916,E2 -897.2455} C_DIS
LIN {X -0.7176,Y -35.3271,Z 62,A -97.0927,B 24.8567,C -2.762,E1 24.9988,E2 -899.8171} C_DIS
LIN {X -0.7176,Y -35.3271,Z 62,A -97.0927,B 24.8567,C -2.762,E1 24.9988,E2 -899.8171} C_DIS
Enddeposition()
LIN {X 0.1856,Y -34.3479,Z 62,A -95.3197,B 24.8545,C -2.7829,E1 25.0039,E2 -901.6397} C_DIS
Startdeposition()
$VEL.CP = VEL_PRINT
LIN {X -0.8177,Y -34.3452,Z 62,A -98.5892,B 24.8565,C -2.7636,E1 24.9946,E2 -898.3243} C_DIS
LIN {X -2.7606,Y -34.2436,Z 62,A -101.8201,B 24.8565,C -2.7636,E1 24.9856,E2 -895.0924} C_DIS
LIN {X -4.3992,Y -34.0718,Z 62,A -104.3739,B 24.8563,C -2.7662,E1 24.9785,E2 -892.5431} C_DIS
LIN {X -6.1336,Y -33.8027,Z 62,A -107.5532,B 24.8565,C -2.7642,E1 24.9698,E2 -889.356} C_DIS
LIN {X -7.7885,Y -33.4602,Z 62,A -110.2997,B 24.8563,C -2.7663,E1 24.9623,E2 -886.6111} C_DIS
LIN {X -9.3283,Y -33.0639,Z 62,A -113.0367,B 24.8562,C -2.7669,E1 24.9549,E2 -883.8714} C_DIS
LIN {X -11.2949,Y -32.445,Z 62,A -116.5853,B 24.856,C -2.7684,E1 24.9455,E2 -880.3198} C_DIS
LIN {X -13.152,Y -31.7381,Z 62,A -119.7184,B 24.8555,C -2.7734,E1 24.9373,E2 -877.1918} C_DIS
LIN {X -15.2574,Y -30.7808,Z 62,A -124.3237,B 24.8559,C -2.7702,E1 24.9257,E2 -872.567} C_DIS
LIN {X -17.1298,Y -29.7794,Z 62,A -127.7798,B 24.8553,C -2.7758,E1 24.9173,E2 -869.1142} C_DIS
LIN {X -19.5074,Y -28.2793,Z 62,A -131.8679,B 24.8539,C -2.7888,E1 24.9078,E2 -865.0438} C_DIS
LIN {X -21.1461,Y -27.0762,Z 62,A -135.6132,B 24.8537,C -2.7912,E1 24.8994,E2 -861.2907} C_DIS
LIN {X -22.9226,Y -25.589,Z 62,A -139.2684,B 24.8527,C -2.8004,E1 24.8917,E2 -857.6433} C_DIS
LIN {X -24.5866,Y -23.9946,Z 62,A -143.3527,B 24.8521,C -2.806,E1 24.8836,E2 -853.5552} C_DIS
LIN {X -26.2043,Y -22.2168,Z 62,A -147.4637,B 24.8513,C -2.8139,E1 24.876,E2 -849.4446} C_DIS
LIN {X -27.6806,Y -20.3478,Z 62,A -151.5788,B 24.8504,C -2.822,E1 24.8691,E2 -845.3292} C_DIS
LIN {X -28.7555,Y -18.7985,Z 62,A -154.2929,B 24.8492,C -2.8336,E1 24.8649,E2 -842.6293} C_DIS
LIN {X -29.6664,Y -17.3248,Z 62,A -157.3182,B 24.8485,C -2.8398,E1 24.8605,E2 -839.6033} C_DIS
LIN {X -30.5442,Y -15.726,Z 62,A -160.1319,B 24.8474,C -2.8499,E1 24.8569,E2 -836.7987} C_DIS
LIN {X -31.3644,Y -14.0186,Z 62,A -164.1453,B 24.8473,C -2.8513,E1 24.8522,E2 -832.7668} C_DIS
LIN {X -32.7042,Y -10.5207,Z 62,A -170.3932,B 24.8453,C -2.8693,E1 24.8463,E2 -826.5264} C_DIS
LIN {X -33.491,Y -7.6551,Z 62,A -174.4726,B 24.8429,C -2.8913,E1 24.8435,E2 -822.4759} C_DIS
LIN {X -33.75,Y -6.4175,Z 62,A -176.777,B 24.8424,C -2.896,E1 24.8423,E2 -820.1692} C_DIS
LIN {X -34.0057,Y -4.8844,Z 62,A -179.7284,B 24.8419,C -2.901,E1 24.841,E2 -817.2122} C_DIS
LIN {X -34.2914,Y -2.0941,Z 62,A 174.7497,B 24.841,C -2.9087,E1 24.8398,E2 -811.6756} C_DIS
LIN {X -34.2939,Y 2.0477,Z 62,A 169.2404,B 24.8374,C -2.9416,E1 24.8401,E2 -806.2118} C_DIS
LIN {X -34.0927,Y 4.2372,Z 62,A 164.3169,B 24.8372,C -2.9429,E1 24.8416,E2 -801.262} C_DIS
LIN {X -33.4413,Y 7.8676,Z 62,A 158.6962,B 24.8346,C -2.9663,E1 24.8447,E2 -795.6642} C_DIS
LIN {X -32.9688,Y 9.659,Z 62,A 156.0603,B 24.8332,C -2.9795,E1 24.8467,E2 -793.0445} C_DIS
LIN {X -32.61,Y 10.8101,Z 62,A 152.9706,B 24.8335,C -2.9768,E1 24.8494,E2 -789.9306} C_DIS
LIN {X -31.2599,Y 14.2507,Z 62,A 147.6639,B 24.8306,C -3.002,E1 24.8551,E2 -784.655} C_DIS
LIN {X -30.486,Y 15.8388,Z 62,A 144.4322,B 24.8299,C -3.0081,E1 24.8592,E2 -781.4206} C_DIS
LIN {X -29.1991,Y 18.1017,Z 62,A 139.0558,B 24.8295,C -3.0116,E1 24.8669,E2 -776.0248} C_DIS
LIN {X -26.6304,Y 21.7042,Z 62,A 133.0379,B 24.826,C -3.0426,E1 24.8769,E2 -770.052} C_DIS
LIN {X -25.7492,Y 22.7432,Z 62,A 129.8907,B 24.8262,C -3.0406,E1 24.8828,E2 -766.8859} C_DIS
LIN {X -23.3353,Y 25.2133,Z 62,A 124.9288,B 24.8239,C -3.0611,E1 24.8925,E2 -761.9521} C_DIS
Enddeposition()
END
